LIN {X 0.048,Y -167.704,Z 705.356,A 0.000,B 0.000,C 90.000,E1 244.101} C_DIS
LIN {X 0.061,Y -166.391,Z 705.347,A 0.000,B 0.000,C 90.000,E1 242.359} C_DIS
LIN {X 0.052,Y -163.118,Z 705.327,A 0.000,B 0.000,C 90.000,E1 238.869} C_DIS
LIN {X 0.102,Y -161.067,Z 705.313,A 0.000,B 0.000,C 90.000,E1 236.215} C_DIS
LIN {X -0.010,Y -157.800,Z 705.293,A 0.000,B 0.000,C 90.000,E1 232.718} C_DIS
LIN {X -0.072,Y -155.836,Z 705.278,A 0.000,B 0.000,C 90.000,E1 230.070} C_DIS
LIN {X -0.015,Y -152.086,Z 705.253,A 0.000,B 0.000,C 90.000,E1 225.567} C_DIS
LIN {X 0.004,Y -150.337,Z 705.238,A 0.000,B 0.000,C 90.000,E1 222.852} C_DIS
LIN {X 0.025,Y -147.076,Z 705.213,A 0.000,B 0.000,C 90.000,E1 218.302} C_DIS
LIN {X -0.071,Y -145.650,Z 705.198,A 0.000,B 0.000,C 90.000,E1 215.598} C_DIS
LIN {X -0.067,Y -143.032,Z 705.172,A 0.000,B 0.000,C 90.000,E1 211.003} C_DIS
LIN {X 0.059,Y -141.657,Z 705.152,A 0.000,B 0.000,C 90.000,E1 207.257} C_DIS
LIN {X -0.022,Y -139.447,Z 705.115,A 0.000,B 0.000,C 90.000,E1 200.791} C_DIS
LIN {X 0.031,Y -139.180,Z 705.105,A 0.000,B 0.000,C 90.000,E1 198.906} C_DIS
LIN {X 0.059,Y -138.320,Z 705.053,A 0.000,B 0.000,C 90.000,E1 189.557} C_DIS
LIN {X 0.069,Y -139.465,Z 705.007,A 0.000,B 0.000,C 90.000,E1 181.146} C_DIS
LIN {X 0.010,Y -141.029,Z 704.975,A 0.000,B 0.000,C 90.000,E1 175.584} C_DIS
LIN {X -0.036,Y -142.396,Z 704.960,A 0.000,B 0.000,C 90.000,E1 172.818} C_DIS
LIN {X 0.026,Y -144.628,Z 704.934,A 0.000,B 0.000,C 90.000,E1 168.173} C_DIS
LIN {X -0.055,Y -147.823,Z 704.909,A 0.000,B 0.000,C 90.000,E1 163.614} C_DIS
LIN {X 0.031,Y -150.514,Z 704.889,A 0.000,B 0.000,C 90.000,E1 159.934} C_DIS
LIN {X 0.052,Y -153.976,Z 704.868,A 0.000,B 0.000,C 90.000,E1 156.305} C_DIS
LIN {X -0.027,Y -157.387,Z 704.849,A 0.000,B 0.000,C 90.000,E1 152.743} C_DIS
LIN {X -0.085,Y -161.592,Z 704.829,A 0.000,B 0.000,C 90.000,E1 149.203} C_DIS
LIN {X -0.075,Y -165.789,Z 704.809,A 0.000,B 0.000,C 90.000,E1 145.674} C_DIS
LIN {X -0.089,Y -170.750,Z 704.790,A 0.000,B 0.000,C 90.000,E1 142.190} C_DIS
LIN {X 0.069,Y -175.622,Z 704.771,A 0.000,B 0.000,C 90.000,E1 138.690} C_DIS
LIN {X -0.062,Y -181.238,Z 704.752,A 0.000,B 0.000,C 90.000,E1 135.324} C_DIS
LIN {X 0.069,Y -186.708,Z 704.733,A 0.000,B 0.000,C 90.000,E1 131.919} C_DIS
LIN {X 0.013,Y -191.370,Z 704.719,A 0.000,B 0.000,C 90.000,E1 129.402} C_DIS
LIN {X -0.035,Y -289.460,Z 704.719,A 0.000,B 0.000,C 90.000,E1 129.402} C_DIS
LIN {X 0.082,Y -291.032,Z 704.719,A 0.000,B 0.000,C 90.000,E1 129.358} C_DIS
LIN {X -0.059,Y -295.409,Z 704.718,A 0.000,B 0.000,C 90.000,E1 129.197} C_DIS
LIN {X 0.028,Y -297.779,Z 704.717,A 0.000,B 0.000,C 90.000,E1 128.991} C_DIS
LIN {X -0.027,Y -301.000,Z 704.715,A 0.000,B 0.000,C 90.000,E1 128.624} C_DIS
LIN {X -0.016,Y -302.956,Z 704.713,A 0.000,B 0.000,C 90.000,E1 128.302} C_DIS
LIN {X 0.045,Y -304.482,Z 704.711,A 0.000,B 0.000,C 90.000,E1 127.971} C_DIS
LIN {X 0.006,Y -305.724,Z 704.709,A 0.000,B 0.000,C 90.000,E1 127.649} C_DIS
LIN {X 0.198,Y -317.437,Z 704.687,A 0.000,B 0.000,C 90.000,E1 123.706} C_DIS
LIN {X -0.041,Y -327.590,Z 704.672,A 0.000,B 0.000,C 90.000,E1 120.875} C_DIS
LIN {X 0.128,Y -339.075,Z 704.656,A 0.000,B 0.000,C 90.000,E1 118.025} C_DIS
LIN {X -0.014,Y -352.001,Z 704.640,A 0.000,B 0.000,C 90.000,E1 115.283} C_DIS
LIN {X -0.151,Y -364.788,Z 704.627,A 0.000,B 0.000,C 90.000,E1 112.898} C_DIS
LIN {X 0.230,Y -378.895,Z 704.614,A 0.000,B 0.000,C 90.000,E1 110.482} C_DIS
LIN {X -0.150,Y -394.422,Z 704.601,A 0.000,B 0.000,C 90.000,E1 108.236} C_DIS
LIN {X -0.016,Y -411.481,Z 704.589,A 0.000,B 0.000,C 90.000,E1 105.969} C_DIS
LIN {X 0.046,Y -430.198,Z 704.577,A 0.000,B 0.000,C 90.000,E1 103.772} C_DIS
LIN {X -0.104,Y -450.192,Z 704.565,A 0.000,B 0.000,C 90.000,E1 101.715} C_DIS
LIN {X 0.076,Y -468.132,Z 704.556,A 0.000,B 0.000,C 90.000,E1 100.018} C_DIS
LIN {X 0.038,Y -470.302,Z 704.554,A 0.000,B 0.000,C 90.000,E1 99.792} C_DIS
LIN {X -0.111,Y -472.091,Z 704.553,A 0.000,B 0.000,C 90.000,E1 99.557} C_DIS
LIN {X 0.203,Y -473.434,Z 704.552,A 0.000,B 0.000,C 90.000,E1 99.265} C_DIS
LIN {X -0.154,Y -475.119,Z 704.549,A 0.000,B 0.000,C 90.000,E1 98.803} C_DIS
LIN {X 0.036,Y -475.734,Z 704.546,A 0.000,B 0.000,C 90.000,E1 98.276} C_DIS
LIN {X 0.167,Y -475.383,Z 704.543,A 0.000,B 0.000,C 90.000,E1 97.757} C_DIS
LIN {X -0.170,Y -474.017,Z 704.540,A 0.000,B 0.000,C 90.000,E1 97.296} C_DIS
LIN {X 0.104,Y -472.884,Z 704.539,A 0.000,B 0.000,C 90.000,E1 97.011} C_DIS
LIN {X -0.182,Y -469.662,Z 704.536,A 0.000,B 0.000,C 90.000,E1 96.543} C_DIS
LIN {X -0.116,Y -451.783,Z 704.521,A 0.000,B 0.000,C 90.000,E1 93.726} C_DIS
LIN {X 0.073,Y -437.091,Z 704.506,A 0.000,B 0.000,C 90.000,E1 91.088} C_DIS
LIN {X 0.141,Y -428.050,Z 704.497,A 0.000,B 0.000,C 90.000,E1 89.484} C_DIS
LIN {X 0.059,Y -418.745,Z 704.488,A 0.000,B 0.000,C 90.000,E1 87.879} C_DIS
LIN {X -0.107,Y -407.783,Z 704.478,A 0.000,B 0.000,C 90.000,E1 85.988} C_DIS
LIN {X -0.039,Y -396.834,Z 704.467,A 0.000,B 0.000,C 90.000,E1 84.033} C_DIS
LIN {X -0.045,Y -381.422,Z 704.451,A 0.000,B 0.000,C 90.000,E1 81.197} C_DIS
LIN {X 0.006,Y -368.132,Z 704.437,A 0.000,B 0.000,C 90.000,E1 78.578} C_DIS
LIN {X -0.201,Y -353.954,Z 704.420,A 0.000,B 0.000,C 90.000,E1 75.644} C_DIS
LIN {X -0.131,Y -340.345,Z 704.403,A 0.000,B 0.000,C 90.000,E1 72.598} C_DIS
LIN {X -0.098,Y -329.846,Z 704.389,A 0.000,B 0.000,C 90.000,E1 70.115} C_DIS
LIN {X 0.087,Y -317.557,Z 704.372,A 0.000,B 0.000,C 90.000,E1 66.922} C_DIS
LIN {X 0.085,Y -307.850,Z 704.356,A 0.000,B 0.000,C 90.000,E1 64.024} C_DIS
LIN {X -0.151,Y -298.135,Z 704.338,A 0.000,B 0.000,C 90.000,E1 60.795} C_DIS
LIN {X -0.097,Y -289.035,Z 704.319,A 0.000,B 0.000,C 90.000,E1 57.454} C_DIS
LIN {X -0.026,Y -282.114,Z 704.304,A 0.000,B 0.000,C 90.000,E1 54.736} C_DIS
LIN {X -0.020,Y -277.046,Z 704.293,A 0.000,B 0.000,C 90.000,E1 52.683} C_DIS
LIN {X 0.048,Y -271.812,Z 704.281,A 0.000,B 0.000,C 90.000,E1 50.598} C_DIS
LIN {X -0.057,Y -266.456,Z 704.270,A 0.000,B 0.000,C 90.000,E1 48.528} C_DIS
LIN {X 0.116,Y -260.753,Z 704.258,A 0.000,B 0.000,C 90.000,E1 46.377} C_DIS
LIN {X -0.019,Y -254.912,Z 704.246,A 0.000,B 0.000,C 90.000,E1 44.271} C_DIS
LIN {X 0.105,Y -248.878,Z 704.234,A 0.000,B 0.000,C 90.000,E1 42.081} C_DIS
LIN {X -0.052,Y -242.729,Z 704.222,A 0.000,B 0.000,C 90.000,E1 39.930} C_DIS
LIN {X -0.017,Y -232.750,Z 704.201,A 0.000,B 0.000,C 90.000,E1 36.217} C_DIS
LIN {X 0.054,Y -223.570,Z 704.180,A 0.000,B 0.000,C 90.000,E1 32.418} C_DIS
LIN {X 0.088,Y -216.951,Z 704.163,A 0.000,B 0.000,C 90.000,E1 29.333} C_DIS
LIN {X 0.021,Y -211.168,Z 704.146,A 0.000,B 0.000,C 90.000,E1 26.232} C_DIS
LIN {X 0.009,Y -206.116,Z 704.128,A 0.000,B 0.000,C 90.000,E1 23.078} C_DIS
LIN {X 0.001,Y -200.975,Z 704.106,A 0.000,B 0.000,C 90.000,E1 19.087} C_DIS
LIN {X -0.045,Y -197.005,Z 704.084,A 0.000,B 0.000,C 90.000,E1 15.064} C_DIS
LIN {X 0.079,Y -193.660,Z 704.056,A 0.000,B 0.000,C 90.000,E1 10.141} C_DIS
LIN {X 0.021,Y -191.501,Z 704.011,A 0.000,B 0.000,C 90.000,E1 1.949} C_DIS
LIN {X -0.072,Y -193.432,Z 703.965,A 0.000,B 0.000,C 90.000,E1 353.799} C_DIS
LIN {X -0.003,Y -196.450,Z 703.938,A 0.000,B 0.000,C 90.000,E1 348.870} C_DIS
LIN {X -0.015,Y -200.116,Z 703.916,A 0.000,B 0.000,C 90.000,E1 344.810} C_DIS
LIN {X -0.030,Y -204.725,Z 703.893,A 0.000,B 0.000,C 90.000,E1 340.786} C_DIS
LIN {X -0.012,Y -210.168,Z 703.871,A 0.000,B 0.000,C 90.000,E1 336.794} C_DIS
LIN {X -0.073,Y -216.346,Z 703.849,A 0.000,B 0.000,C 90.000,E1 332.871} C_DIS
LIN {X 0.070,Y -223.240,Z 703.828,A 0.000,B 0.000,C 90.000,E1 328.948} C_DIS
LIN {X 0.008,Y -230.745,Z 703.806,A 0.000,B 0.000,C 90.000,E1 325.135} C_DIS
LIN {X -0.035,Y -238.853,Z 703.785,A 0.000,B 0.000,C 90.000,E1 321.376} C_DIS
LIN {X 0.120,Y -247.875,Z 703.765,A 0.000,B 0.000,C 90.000,E1 317.634} C_DIS
LIN {X -0.006,Y -257.951,Z 703.745,A 0.000,B 0.000,C 90.000,E1 314.028} C_DIS
LIN {X 0.048,Y -269.153,Z 703.725,A 0.000,B 0.000,C 90.000,E1 310.458} C_DIS
LIN {X 0.082,Y -280.335,Z 703.707,A 0.000,B 0.000,C 90.000,E1 307.317} C_DIS
LIN {X 0.085,Y -294.112,Z 703.688,A 0.000,B 0.000,C 90.000,E1 303.913} C_DIS
LIN {X 0.115,Y -309.286,Z 703.670,A 0.000,B 0.000,C 90.000,E1 300.590} C_DIS
LIN {X -0.011,Y -322.591,Z 703.656,A 0.000,B 0.000,C 90.000,E1 298.025} C_DIS
LIN {X -0.155,Y -340.634,Z 703.638,A 0.000,B 0.000,C 90.000,E1 294.899} C_DIS
LIN {X 0.090,Y -356.064,Z 703.625,A 0.000,B 0.000,C 90.000,E1 292.408} C_DIS
LIN {X -0.208,Y -372.171,Z 703.611,A 0.000,B 0.000,C 90.000,E1 290.066} C_DIS
LIN {X 0.112,Y -390.115,Z 703.598,A 0.000,B 0.000,C 90.000,E1 287.692} C_DIS
LIN {X -0.117,Y -404.103,Z 703.589,A 0.000,B 0.000,C 90.000,E1 286.024} C_DIS
LIN {X -0.100,Y -417.902,Z 703.580,A 0.000,B 0.000,C 90.000,E1 284.356} C_DIS
LIN {X -0.206,Y -429.223,Z 703.572,A 0.000,B 0.000,C 90.000,E1 283.008} C_DIS
LIN {X 0.093,Y -437.971,Z 703.566,A 0.000,B 0.000,C 90.000,E1 281.895} C_DIS
LIN {X -0.136,Y -448.227,Z 703.559,A 0.000,B 0.000,C 90.000,E1 280.602} C_DIS
LIN {X -0.022,Y -464.309,Z 703.547,A 0.000,B 0.000,C 90.000,E1 278.511} C_DIS
LIN {X 0.115,Y -472.091,Z 703.542,A 0.000,B 0.000,C 90.000,E1 277.473} C_DIS
LIN {X 0.074,Y -477.214,Z 703.537,A 0.000,B 0.000,C 90.000,E1 276.720} C_DIS
LIN {X 0.213,Y -480.183,Z 703.535,A 0.000,B 0.000,C 90.000,E1 276.201} C_DIS
LIN {X -0.110,Y -482.767,Z 703.532,A 0.000,B 0.000,C 90.000,E1 275.739} C_DIS
LIN {X 0.061,Y -484.885,Z 703.529,A 0.000,B 0.000,C 90.000,E1 275.220} C_DIS
LIN {X 0.246,Y -486.541,Z 703.526,A 0.000,B 0.000,C 90.000,E1 274.702} C_DIS
LIN {X -0.087,Y -487.760,Z 703.523,A 0.000,B 0.000,C 90.000,E1 274.245} C_DIS
LIN {X 0.113,Y -488.620,Z 703.521,A 0.000,B 0.000,C 90.000,E1 273.726} C_DIS
LIN {X -0.200,Y -489.020,Z 703.518,A 0.000,B 0.000,C 90.000,E1 273.269} C_DIS
LIN {X 0.008,Y -489.135,Z 703.515,A 0.000,B 0.000,C 90.000,E1 272.751} C_DIS
LIN {X 0.194,Y -488.868,Z 703.513,A 0.000,B 0.000,C 90.000,E1 272.236} C_DIS
LIN {X -0.089,Y -488.311,Z 703.510,A 0.000,B 0.000,C 90.000,E1 271.776} C_DIS
LIN {X 0.096,Y -487.341,Z 703.507,A 0.000,B 0.000,C 90.000,E1 271.260} C_DIS
LIN {X -0.207,Y -485.976,Z 703.504,A 0.000,B 0.000,C 90.000,E1 270.802} C_DIS
LIN {X -0.028,Y -484.154,Z 703.502,A 0.000,B 0.000,C 90.000,E1 270.286} C_DIS
LIN {X 0.143,Y -481.763,Z 703.499,A 0.000,B 0.000,C 90.000,E1 269.771} C_DIS
LIN {X -0.184,Y -478.781,Z 703.496,A 0.000,B 0.000,C 90.000,E1 269.312} C_DIS
LIN {X -0.048,Y -474.923,Z 703.493,A 0.000,B 0.000,C 90.000,E1 268.797} C_DIS
LIN {X 0.066,Y -470.084,Z 703.490,A 0.000,B 0.000,C 90.000,E1 268.282} C_DIS
LIN {X -0.053,Y -467.317,Z 703.489,A 0.000,B 0.000,C 90.000,E1 268.051} C_DIS
LIN {X -0.029,Y -461.152,Z 703.487,A 0.000,B 0.000,C 90.000,E1 267.593} C_DIS
LIN {X 0.122,Y -457.794,Z 703.485,A 0.000,B 0.000,C 90.000,E1 267.364} C_DIS
LIN {X 0.064,Y -454.502,Z 703.484,A 0.000,B 0.000,C 90.000,E1 267.192} C_DIS
LIN {X -0.179,Y -447.359,Z 703.483,A 0.000,B 0.000,C 90.000,E1 266.906} C_DIS
LIN {X 0.142,Y -440.044,Z 703.481,A 0.000,B 0.000,C 90.000,E1 266.617} C_DIS
LIN {X -0.018,Y -431.920,Z 703.480,A 0.000,B 0.000,C 90.000,E1 266.445} C_DIS
LIN {X -0.208,Y -426.165,Z 703.480,A 0.000,B 0.000,C 90.000,E1 266.388} C_DIS
LIN {X 0.159,Y -417.344,Z 703.479,A 0.000,B 0.000,C 90.000,E1 266.274} C_DIS
LIN {X 0.048,Y -180.934,Z 703.479,A 0.000,B 0.000,C 90.000,E1 266.274} C_DIS
LIN {X 0.080,Y -180.714,Z 703.470,A 0.000,B 0.000,C 90.000,E1 264.552} C_DIS
LIN {X -0.002,Y -178.800,Z 703.442,A 0.000,B 0.000,C 90.000,E1 259.511} C_DIS
LIN {X 0.075,Y -175.846,Z 703.413,A 0.000,B 0.000,C 90.000,E1 254.393} C_DIS
LIN {X 0.075,Y -172.037,Z 703.385,A 0.000,B 0.000,C 90.000,E1 249.263} C_DIS
LIN {X 0.051,Y -171.469,Z 703.380,A 0.000,B 0.000,C 90.000,E1 248.411} C_DIS
LIN {X 0.030,Y -167.700,Z 703.356,A 0.000,B 0.000,C 90.000,E1 244.101} C_DIS
LIN {X 0.043,Y -166.385,Z 703.346,A 0.000,B 0.000,C 90.000,E1 242.359} C_DIS
LIN {X 0.035,Y -163.113,Z 703.327,A 0.000,B 0.000,C 90.000,E1 238.869} C_DIS
LIN {X 0.085,Y -161.062,Z 703.313,A 0.000,B 0.000,C 90.000,E1 236.215} C_DIS
LIN {X -0.027,Y -157.795,Z 703.293,A 0.000,B 0.000,C 90.000,E1 232.718} C_DIS
LIN {X 0.012,Y -155.832,Z 703.278,A 0.000,B 0.000,C 90.000,E1 230.033} C_DIS
LIN {X -0.031,Y -152.082,Z 703.253,A 0.000,B 0.000,C 90.000,E1 225.567} C_DIS
LIN {X -0.013,Y -150.333,Z 703.238,A 0.000,B 0.000,C 90.000,E1 222.852} C_DIS
LIN {X 0.008,Y -147.073,Z 703.213,A 0.000,B 0.000,C 90.000,E1 218.302} C_DIS
LIN {X -0.088,Y -145.647,Z 703.198,A 0.000,B 0.000,C 90.000,E1 215.598} C_DIS
LIN {X -0.083,Y -143.029,Z 703.172,A 0.000,B 0.000,C 90.000,E1 211.003} C_DIS
LIN {X 0.044,Y -141.655,Z 703.152,A 0.000,B 0.000,C 90.000,E1 207.257} C_DIS
LIN {X -0.037,Y -139.445,Z 703.115,A 0.000,B 0.000,C 90.000,E1 200.791} C_DIS
LIN {X 0.016,Y -139.179,Z 703.105,A 0.000,B 0.000,C 90.000,E1 198.906} C_DIS
LIN {X 0.044,Y -138.320,Z 703.053,A 0.000,B 0.000,C 90.000,E1 189.557} C_DIS
LIN {X 0.053,Y -139.467,Z 703.006,A 0.000,B 0.000,C 90.000,E1 181.146} C_DIS
LIN {X -0.006,Y -141.032,Z 702.975,A 0.000,B 0.000,C 90.000,E1 175.584} C_DIS
LIN {X -0.052,Y -142.399,Z 702.960,A 0.000,B 0.000,C 90.000,E1 172.818} C_DIS
LIN {X 0.011,Y -144.631,Z 702.934,A 0.000,B 0.000,C 90.000,E1 168.173} C_DIS
LIN {X 0.071,Y -147.827,Z 702.909,A 0.000,B 0.000,C 90.000,E1 163.559} C_DIS
LIN {X 0.016,Y -150.520,Z 702.889,A 0.000,B 0.000,C 90.000,E1 159.934} C_DIS
LIN {X 0.035,Y -153.982,Z 702.868,A 0.000,B 0.000,C 90.000,E1 156.305} C_DIS
LIN {X -0.045,Y -157.394,Z 702.849,A 0.000,B 0.000,C 90.000,E1 152.743} C_DIS
LIN {X 0.036,Y -161.600,Z 702.829,A 0.000,B 0.000,C 90.000,E1 149.154} C_DIS
LIN {X -0.092,Y -165.796,Z 702.809,A 0.000,B 0.000,C 90.000,E1 145.674} C_DIS
LIN {X 0.028,Y -170.759,Z 702.790,A 0.000,B 0.000,C 90.000,E1 142.145} C_DIS
LIN {X 0.051,Y -175.632,Z 702.771,A 0.000,B 0.000,C 90.000,E1 138.690} C_DIS
LIN {X -0.080,Y -181.247,Z 702.752,A 0.000,B 0.000,C 90.000,E1 135.324} C_DIS
LIN {X 0.050,Y -186.718,Z 702.733,A 0.000,B 0.000,C 90.000,E1 131.919} C_DIS
LIN {X 0.053,Y -191.351,Z 702.719,A 0.000,B 0.000,C 90.000,E1 129.402} C_DIS
LIN {X 0.044,Y -289.167,Z 702.719,A 0.000,B 0.000,C 90.000,E1 129.402} C_DIS
LIN {X 0.053,Y -291.778,Z 702.719,A 0.000,B 0.000,C 90.000,E1 129.358} C_DIS
LIN {X -0.089,Y -295.650,Z 702.718,A 0.000,B 0.000,C 90.000,E1 129.197} C_DIS
LIN {X -0.002,Y -297.932,Z 702.717,A 0.000,B 0.000,C 90.000,E1 128.991} C_DIS
LIN {X -0.058,Y -301.080,Z 702.715,A 0.000,B 0.000,C 90.000,E1 128.624} C_DIS
LIN {X -0.074,Y -303.031,Z 702.713,A 0.000,B 0.000,C 90.000,E1 128.302} C_DIS
LIN {X -0.040,Y -304.551,Z 702.711,A 0.000,B 0.000,C 90.000,E1 127.971} C_DIS
LIN {X -0.081,Y -305.766,Z 702.709,A 0.000,B 0.000,C 90.000,E1 127.649} C_DIS
LIN {X 0.109,Y -317.469,Z 702.687,A 0.000,B 0.000,C 90.000,E1 123.706} C_DIS
LIN {X -0.131,Y -327.628,Z 702.671,A 0.000,B 0.000,C 90.000,E1 120.875} C_DIS
LIN {X 0.035,Y -339.121,Z 702.656,A 0.000,B 0.000,C 90.000,E1 118.025} C_DIS
LIN {X -0.107,Y -352.054,Z 702.640,A 0.000,B 0.000,C 90.000,E1 115.283} C_DIS
LIN {X 0.088,Y -364.850,Z 702.627,A 0.000,B 0.000,C 90.000,E1 112.845} C_DIS
LIN {X 0.132,Y -378.965,Z 702.614,A 0.000,B 0.000,C 90.000,E1 110.482} C_DIS
LIN {X 0.124,Y -394.501,Z 702.601,A 0.000,B 0.000,C 90.000,E1 108.181} C_DIS
LIN {X -0.119,Y -411.570,Z 702.589,A 0.000,B 0.000,C 90.000,E1 105.969} C_DIS
LIN {X -0.060,Y -430.298,Z 702.576,A 0.000,B 0.000,C 90.000,E1 103.772} C_DIS
LIN {X -0.206,Y -450.295,Z 702.565,A 0.000,B 0.000,C 90.000,E1 101.715} C_DIS
LIN {X -0.023,Y -468.237,Z 702.556,A 0.000,B 0.000,C 90.000,E1 100.018} C_DIS
LIN {X -0.061,Y -470.396,Z 702.554,A 0.000,B 0.000,C 90.000,E1 99.792} C_DIS
LIN {X -0.211,Y -472.176,Z 702.553,A 0.000,B 0.000,C 90.000,E1 99.557} C_DIS
LIN {X 0.104,Y -473.513,Z 702.552,A 0.000,B 0.000,C 90.000,E1 99.265} C_DIS
LIN {X -0.253,Y -475.188,Z 702.549,A 0.000,B 0.000,C 90.000,E1 98.803} C_DIS
LIN {X -0.062,Y -475.795,Z 702.546,A 0.000,B 0.000,C 90.000,E1 98.276} C_DIS
LIN {X 0.069,Y -475.436,Z 702.543,A 0.000,B 0.000,C 90.000,E1 97.757} C_DIS
LIN {X 0.203,Y -474.060,Z 702.540,A 0.000,B 0.000,C 90.000,E1 97.239} C_DIS
LIN {X 0.064,Y -472.922,Z 702.539,A 0.000,B 0.000,C 90.000,E1 97.004} C_DIS
LIN {X 0.188,Y -469.694,Z 702.536,A 0.000,B 0.000,C 90.000,E1 96.486} C_DIS
LIN {X -0.208,Y -451.768,Z 702.521,A 0.000,B 0.000,C 90.000,E1 93.726} C_DIS
LIN {X -0.016,Y -437.088,Z 702.506,A 0.000,B 0.000,C 90.000,E1 91.088} C_DIS
LIN {X 0.054,Y -428.082,Z 702.497,A 0.000,B 0.000,C 90.000,E1 89.484} C_DIS
LIN {X 0.081,Y -417.200,Z 702.487,A 0.000,B 0.000,C 90.000,E1 87.593} C_DIS
LIN {X -0.089,Y -406.241,Z 702.476,A 0.000,B 0.000,C 90.000,E1 85.698} C_DIS
LIN {X -0.118,Y -396.864,Z 702.467,A 0.000,B 0.000,C 90.000,E1 84.033} C_DIS
LIN {X -0.120,Y -381.467,Z 702.451,A 0.000,B 0.000,C 90.000,E1 81.197} C_DIS
LIN {X -0.065,Y -368.205,Z 702.436,A 0.000,B 0.000,C 90.000,E1 78.578} C_DIS
LIN {X 0.075,Y -354.027,Z 702.420,A 0.000,B 0.000,C 90.000,E1 75.589} C_DIS
LIN {X 0.131,Y -340.470,Z 702.403,A 0.000,B 0.000,C 90.000,E1 72.543} C_DIS
LIN {X 0.155,Y -329.993,Z 702.389,A 0.000,B 0.000,C 90.000,E1 70.061} C_DIS
LIN {X 0.038,Y -317.748,Z 702.372,A 0.000,B 0.000,C 90.000,E1 66.922} C_DIS
LIN {X 0.042,Y -308.053,Z 702.356,A 0.000,B 0.000,C 90.000,E1 64.024} C_DIS
LIN {X -0.187,Y -298.358,Z 702.338,A 0.000,B 0.000,C 90.000,E1 60.795} C_DIS
LIN {X -0.124,Y -289.286,Z 702.319,A 0.000,B 0.000,C 90.000,E1 57.454} C_DIS
LIN {X -0.046,Y -282.387,Z 702.304,A 0.000,B 0.000,C 90.000,E1 54.736} C_DIS
LIN {X -0.036,Y -277.320,Z 702.293,A 0.000,B 0.000,C 90.000,E1 52.683} C_DIS
LIN {X 0.038,Y -272.122,Z 702.281,A 0.000,B 0.000,C 90.000,E1 50.598} C_DIS
LIN {X -0.060,Y -266.768,Z 702.270,A 0.000,B 0.000,C 90.000,E1 48.528} C_DIS
LIN {X 0.118,Y -261.057,Z 702.258,A 0.000,B 0.000,C 90.000,E1 46.377} C_DIS
LIN {X -0.012,Y -255.182,Z 702.246,A 0.000,B 0.000,C 90.000,E1 44.271} C_DIS
LIN {X -0.067,Y -249.164,Z 702.234,A 0.000,B 0.000,C 90.000,E1 42.123} C_DIS
LIN {X -0.034,Y -242.980,Z 702.222,A 0.000,B 0.000,C 90.000,E1 39.930} C_DIS
LIN {X 0.006,Y -232.950,Z 702.201,A 0.000,B 0.000,C 90.000,E1 36.217} C_DIS
LIN {X 0.082,Y -223.756,Z 702.180,A 0.000,B 0.000,C 90.000,E1 32.418} C_DIS
LIN {X 0.121,Y -217.115,Z 702.163,A 0.000,B 0.000,C 90.000,E1 29.333} C_DIS
LIN {X 0.057,Y -211.333,Z 702.146,A 0.000,B 0.000,C 90.000,E1 26.232} C_DIS
LIN {X 0.048,Y -206.277,Z 702.128,A 0.000,B 0.000,C 90.000,E1 23.078} C_DIS
LIN {X 0.044,Y -201.134,Z 702.106,A 0.000,B 0.000,C 90.000,E1 19.087} C_DIS
LIN {X 0.003,Y -197.160,Z 702.084,A 0.000,B 0.000,C 90.000,E1 15.064} C_DIS
LIN {X -0.059,Y -193.825,Z 702.057,A 0.000,B 0.000,C 90.000,E1 10.197} C_DIS
LIN {X 0.082,Y -191.648,Z 702.011,A 0.000,B 0.000,C 90.000,E1 1.949} C_DIS
LIN {X -0.066,Y -193.542,Z 701.965,A 0.000,B 0.000,C 90.000,E1 353.799} C_DIS
LIN {X 0.008,Y -196.562,Z 701.938,A 0.000,B 0.000,C 90.000,E1 348.870} C_DIS
LIN {X -0.001,Y -200.208,Z 701.916,A 0.000,B 0.000,C 90.000,E1 344.810} C_DIS
LIN {X -0.013,Y -204.805,Z 701.893,A 0.000,B 0.000,C 90.000,E1 340.786} C_DIS
LIN {X 0.008,Y -210.234,Z 701.871,A 0.000,B 0.000,C 90.000,E1 336.794} C_DIS
LIN {X -0.050,Y -216.404,Z 701.849,A 0.000,B 0.000,C 90.000,E1 332.871} C_DIS
LIN {X -0.097,Y -223.286,Z 701.828,A 0.000,B 0.000,C 90.000,E1 328.997} C_DIS
LIN {X 0.035,Y -230.773,Z 701.806,A 0.000,B 0.000,C 90.000,E1 325.135} C_DIS
LIN {X -0.006,Y -238.876,Z 701.785,A 0.000,B 0.000,C 90.000,E1 321.376} C_DIS
LIN {X -0.032,Y -247.896,Z 701.765,A 0.000,B 0.000,C 90.000,E1 317.676} C_DIS
LIN {X 0.028,Y -257.967,Z 701.745,A 0.000,B 0.000,C 90.000,E1 314.028} C_DIS
LIN {X 0.084,Y -269.167,Z 701.725,A 0.000,B 0.000,C 90.000,E1 310.458} C_DIS
LIN {X -0.103,Y -280.348,Z 701.707,A 0.000,B 0.000,C 90.000,E1 307.363} C_DIS
LIN {X 0.124,Y -294.121,Z 701.689,A 0.000,B 0.000,C 90.000,E1 303.913} C_DIS
LIN {X 0.157,Y -309.292,Z 701.670,A 0.000,B 0.000,C 90.000,E1 300.590} C_DIS
LIN {X 0.033,Y -322.585,Z 701.656,A 0.000,B 0.000,C 90.000,E1 298.025} C_DIS
LIN {X -0.110,Y -340.598,Z 701.638,A 0.000,B 0.000,C 90.000,E1 294.899} C_DIS
LIN {X -0.155,Y -357.955,Z 701.623,A 0.000,B 0.000,C 90.000,E1 292.153} C_DIS
LIN {X -0.160,Y -372.051,Z 701.611,A 0.000,B 0.000,C 90.000,E1 290.066} C_DIS
LIN {X 0.014,Y -387.646,Z 701.600,A 0.000,B 0.000,C 90.000,E1 288.000} C_DIS
LIN {X -0.146,Y -401.637,Z 701.591,A 0.000,B 0.000,C 90.000,E1 286.315} C_DIS
LIN {X 0.223,Y -415.433,Z 701.581,A 0.000,B 0.000,C 90.000,E1 284.592} C_DIS
LIN {X 0.093,Y -426.792,Z 701.574,A 0.000,B 0.000,C 90.000,E1 283.244} C_DIS
LIN {X -0.057,Y -435.628,Z 701.568,A 0.000,B 0.000,C 90.000,E1 282.187} C_DIS
LIN {X 0.109,Y -446.003,Z 701.560,A 0.000,B 0.000,C 90.000,E1 280.838} C_DIS
LIN {X 0.184,Y -462.066,Z 701.549,A 0.000,B 0.000,C 90.000,E1 278.746} C_DIS
LIN {X -0.102,Y -470.009,Z 701.543,A 0.000,B 0.000,C 90.000,E1 277.757} C_DIS
LIN {X -0.162,Y -475.402,Z 701.539,A 0.000,B 0.000,C 90.000,E1 277.004} C_DIS
LIN {X -0.039,Y -478.609,Z 701.536,A 0.000,B 0.000,C 90.000,E1 276.486} C_DIS
LIN {X -0.083,Y -482.625,Z 701.532,A 0.000,B 0.000,C 90.000,E1 275.739} C_DIS
LIN {X 0.087,Y -484.742,Z 701.529,A 0.000,B 0.000,C 90.000,E1 275.220} C_DIS
LIN {X -0.213,Y -486.412,Z 701.526,A 0.000,B 0.000,C 90.000,E1 274.759} C_DIS
LIN {X -0.063,Y -487.677,Z 701.524,A 0.000,B 0.000,C 90.000,E1 274.245} C_DIS
LIN {X 0.136,Y -488.485,Z 701.521,A 0.000,B 0.000,C 90.000,E1 273.726} C_DIS
LIN {X -0.177,Y -488.916,Z 701.518,A 0.000,B 0.000,C 90.000,E1 273.269} C_DIS
LIN {X 0.030,Y -489.010,Z 701.515,A 0.000,B 0.000,C 90.000,E1 272.751} C_DIS
LIN {X 0.216,Y -488.794,Z 701.513,A 0.000,B 0.000,C 90.000,E1 272.236} C_DIS
LIN {X -0.069,Y -488.232,Z 701.510,A 0.000,B 0.000,C 90.000,E1 271.776} C_DIS
LIN {X 0.117,Y -487.276,Z 701.507,A 0.000,B 0.000,C 90.000,E1 271.260} C_DIS
LIN {X -0.186,Y -485.918,Z 701.504,A 0.000,B 0.000,C 90.000,E1 270.802} C_DIS
LIN {X -0.007,Y -484.089,Z 701.502,A 0.000,B 0.000,C 90.000,E1 270.286} C_DIS
LIN {X 0.162,Y -481.745,Z 701.499,A 0.000,B 0.000,C 90.000,E1 269.771} C_DIS
LIN {X -0.166,Y -478.739,Z 701.496,A 0.000,B 0.000,C 90.000,E1 269.312} C_DIS
LIN {X -0.029,Y -474.902,Z 701.493,A 0.000,B 0.000,C 90.000,E1 268.797} C_DIS
LIN {X 0.084,Y -470.050,Z 701.491,A 0.000,B 0.000,C 90.000,E1 268.282} C_DIS
LIN {X -0.023,Y -467.314,Z 701.489,A 0.000,B 0.000,C 90.000,E1 268.051} C_DIS
LIN {X 0.007,Y -461.260,Z 701.487,A 0.000,B 0.000,C 90.000,E1 267.593} C_DIS
LIN {X 0.156,Y -457.864,Z 701.485,A 0.000,B 0.000,C 90.000,E1 267.364} C_DIS
LIN {X 0.059,Y -450.853,Z 701.483,A 0.000,B 0.000,C 90.000,E1 267.020} C_DIS
LIN {X 0.081,Y -443.504,Z 701.482,A 0.000,B 0.000,C 90.000,E1 266.731} C_DIS
LIN {X 0.125,Y -435.832,Z 701.481,A 0.000,B 0.000,C 90.000,E1 266.502} C_DIS
LIN {X -0.071,Y -431.766,Z 701.480,A 0.000,B 0.000,C 90.000,E1 266.445} C_DIS
LIN {X 0.165,Y -425.980,Z 701.480,A 0.000,B 0.000,C 90.000,E1 266.331} C_DIS
LIN {X 0.107,Y -417.182,Z 701.479,A 0.000,B 0.000,C 90.000,E1 266.274} C_DIS
LIN {X 0.026,Y -180.934,Z 701.479,A 0.000,B 0.000,C 90.000,E1 266.274} C_DIS
LIN {X 0.002,Y -180.906,Z 701.474,A 0.000,B 0.000,C 90.000,E1 265.412} C_DIS
LIN {X 0.059,Y -180.710,Z 701.470,A 0.000,B 0.000,C 90.000,E1 264.552} C_DIS
LIN {X -0.023,Y -178.797,Z 701.442,A 0.000,B 0.000,C 90.000,E1 259.511} C_DIS
LIN {X 0.054,Y -175.843,Z 701.413,A 0.000,B 0.000,C 90.000,E1 254.393} C_DIS
LIN {X 0.053,Y -172.033,Z 701.385,A 0.000,B 0.000,C 90.000,E1 249.263} C_DIS
LIN {X 0.030,Y -171.462,Z 701.380,A 0.000,B 0.000,C 90.000,E1 248.411} C_DIS
LIN {X 0.010,Y -167.694,Z 701.356,A 0.000,B 0.000,C 90.000,E1 244.101} C_DIS
LIN {X 0.024,Y -166.378,Z 701.346,A 0.000,B 0.000,C 90.000,E1 242.359} C_DIS
LIN {X 0.016,Y -163.107,Z 701.327,A 0.000,B 0.000,C 90.000,E1 238.869} C_DIS
LIN {X 0.066,Y -161.054,Z 701.312,A 0.000,B 0.000,C 90.000,E1 236.215} C_DIS
LIN {X 0.048,Y -157.789,Z 701.293,A 0.000,B 0.000,C 90.000,E1 232.683} C_DIS
LIN {X -0.008,Y -155.826,Z 701.278,A 0.000,B 0.000,C 90.000,E1 230.033} C_DIS
LIN {X -0.051,Y -152.077,Z 701.253,A 0.000,B 0.000,C 90.000,E1 225.567} C_DIS
LIN {X -0.032,Y -150.327,Z 701.238,A 0.000,B 0.000,C 90.000,E1 222.852} C_DIS
LIN {X -0.011,Y -147.068,Z 701.213,A 0.000,B 0.000,C 90.000,E1 218.302} C_DIS
LIN {X 0.097,Y -145.643,Z 701.198,A 0.000,B 0.000,C 90.000,E1 215.518} C_DIS
LIN {X 0.094,Y -143.026,Z 701.172,A 0.000,B 0.000,C 90.000,E1 210.924} C_DIS
LIN {X 0.025,Y -141.651,Z 701.151,A 0.000,B 0.000,C 90.000,E1 207.257} C_DIS
LIN {X -0.055,Y -139.444,Z 701.115,A 0.000,B 0.000,C 90.000,E1 200.791} C_DIS
LIN {X -0.003,Y -139.177,Z 701.105,A 0.000,B 0.000,C 90.000,E1 198.906} C_DIS
LIN {X 0.026,Y -138.319,Z 701.053,A 0.000,B 0.000,C 90.000,E1 189.557} C_DIS
LIN {X 0.035,Y -139.468,Z 701.006,A 0.000,B 0.000,C 90.000,E1 181.146} C_DIS
LIN {X -0.025,Y -141.035,Z 700.975,A 0.000,B 0.000,C 90.000,E1 175.584} C_DIS
LIN {X 0.071,Y -142.403,Z 700.960,A 0.000,B 0.000,C 90.000,E1 172.761} C_DIS
LIN {X -0.009,Y -144.636,Z 700.934,A 0.000,B 0.000,C 90.000,E1 168.173} C_DIS
LIN {X 0.052,Y -147.831,Z 700.909,A 0.000,B 0.000,C 90.000,E1 163.559} C_DIS
LIN {X -0.004,Y -150.526,Z 700.888,A 0.000,B 0.000,C 90.000,E1 159.934} C_DIS
LIN {X 0.015,Y -153.988,Z 700.868,A 0.000,B 0.000,C 90.000,E1 156.305} C_DIS
LIN {X -0.064,Y -157.402,Z 700.848,A 0.000,B 0.000,C 90.000,E1 152.743} C_DIS
LIN {X 0.016,Y -161.608,Z 700.829,A 0.000,B 0.000,C 90.000,E1 149.154} C_DIS
LIN {X -0.019,Y -165.805,Z 700.809,A 0.000,B 0.000,C 90.000,E1 145.642} C_DIS
LIN {X 0.007,Y -170.770,Z 700.790,A 0.000,B 0.000,C 90.000,E1 142.145} C_DIS
LIN {X 0.029,Y -175.642,Z 700.771,A 0.000,B 0.000,C 90.000,E1 138.690} C_DIS
LIN {X -0.102,Y -181.256,Z 700.752,A 0.000,B 0.000,C 90.000,E1 135.324} C_DIS
LIN {X 0.028,Y -186.730,Z 700.733,A 0.000,B 0.000,C 90.000,E1 131.919} C_DIS
LIN {X -0.044,Y -191.339,Z 700.719,A 0.000,B 0.000,C 90.000,E1 129.439} C_DIS
LIN {X 0.081,Y -289.525,Z 700.719,A 0.000,B 0.000,C 90.000,E1 129.402} C_DIS
LIN {X 0.019,Y -292.253,Z 700.719,A 0.000,B 0.000,C 90.000,E1 129.358} C_DIS
LIN {X -0.123,Y -295.841,Z 700.718,A 0.000,B 0.000,C 90.000,E1 129.197} C_DIS
LIN {X -0.036,Y -298.058,Z 700.717,A 0.000,B 0.000,C 90.000,E1 128.991} C_DIS
LIN {X -0.093,Y -301.151,Z 700.714,A 0.000,B 0.000,C 90.000,E1 128.624} C_DIS
LIN {X 0.106,Y -303.096,Z 700.713,A 0.000,B 0.000,C 90.000,E1 128.257} C_DIS
LIN {X 0.066,Y -304.610,Z 700.711,A 0.000,B 0.000,C 90.000,E1 127.935} C_DIS
LIN {X 0.081,Y -305.801,Z 700.709,A 0.000,B 0.000,C 90.000,E1 127.604} C_DIS
LIN {X -0.032,Y -316.443,Z 700.689,A 0.000,B 0.000,C 90.000,E1 124.040} C_DIS
LIN {X 0.142,Y -326.464,Z 700.673,A 0.000,B 0.000,C 90.000,E1 121.131} C_DIS
LIN {X -0.181,Y -337.812,Z 700.657,A 0.000,B 0.000,C 90.000,E1 118.359} C_DIS
LIN {X 0.107,Y -350.584,Z 700.642,A 0.000,B 0.000,C 90.000,E1 115.540} C_DIS
LIN {X 0.084,Y -363.228,Z 700.629,A 0.000,B 0.000,C 90.000,E1 113.131} C_DIS
LIN {X -0.062,Y -377.179,Z 700.615,A 0.000,B 0.000,C 90.000,E1 110.791} C_DIS
LIN {X -0.120,Y -392.539,Z 700.603,A 0.000,B 0.000,C 90.000,E1 108.489} C_DIS
LIN {X 0.092,Y -409.418,Z 700.590,A 0.000,B 0.000,C 90.000,E1 106.205} C_DIS
LIN {X 0.106,Y -427.940,Z 700.578,A 0.000,B 0.000,C 90.000,E1 104.008} C_DIS
LIN {X -0.178,Y -447.835,Z 700.566,A 0.000,B 0.000,C 90.000,E1 101.951} C_DIS
LIN {X -0.110,Y -468.325,Z 700.556,A 0.000,B 0.000,C 90.000,E1 100.018} C_DIS
LIN {X -0.147,Y -470.476,Z 700.554,A 0.000,B 0.000,C 90.000,E1 99.792} C_DIS
LIN {X 0.168,Y -472.251,Z 700.553,A 0.000,B 0.000,C 90.000,E1 99.500} C_DIS
LIN {X 0.018,Y -473.584,Z 700.551,A 0.000,B 0.000,C 90.000,E1 99.265} C_DIS
LIN {X 0.131,Y -475.254,Z 700.549,A 0.000,B 0.000,C 90.000,E1 98.746} C_DIS
LIN {X -0.148,Y -475.856,Z 700.546,A 0.000,B 0.000,C 90.000,E1 98.276} C_DIS
LIN {X -0.017,Y -475.493,Z 700.543,A 0.000,B 0.000,C 90.000,E1 97.757} C_DIS
LIN {X 0.119,Y -474.112,Z 700.540,A 0.000,B 0.000,C 90.000,E1 97.239} C_DIS
LIN {X -0.021,Y -472.970,Z 700.539,A 0.000,B 0.000,C 90.000,E1 97.004} C_DIS
LIN {X 0.105,Y -469.738,Z 700.536,A 0.000,B 0.000,C 90.000,E1 96.486} C_DIS
LIN {X 0.163,Y -451.768,Z 700.521,A 0.000,B 0.000,C 90.000,E1 93.669} C_DIS
LIN {X -0.093,Y -437.096,Z 700.506,A 0.000,B 0.000,C 90.000,E1 91.088} C_DIS
LIN {X -0.021,Y -428.119,Z 700.497,A 0.000,B 0.000,C 90.000,E1 89.484} C_DIS
LIN {X 0.008,Y -417.263,Z 700.487,A 0.000,B 0.000,C 90.000,E1 87.593} C_DIS
LIN {X -0.158,Y -406.283,Z 700.476,A 0.000,B 0.000,C 90.000,E1 85.698} C_DIS
LIN {X -0.116,Y -395.327,Z 700.465,A 0.000,B 0.000,C 90.000,E1 83.742} C_DIS
LIN {X -0.155,Y -380.027,Z 700.449,A 0.000,B 0.000,C 90.000,E1 80.905} C_DIS
LIN {X -0.125,Y -368.289,Z 700.436,A 0.000,B 0.000,C 90.000,E1 78.578} C_DIS
LIN {X 0.021,Y -354.111,Z 700.420,A 0.000,B 0.000,C 90.000,E1 75.589} C_DIS
LIN {X 0.082,Y -340.605,Z 700.403,A 0.000,B 0.000,C 90.000,E1 72.543} C_DIS
LIN {X 0.110,Y -330.147,Z 700.389,A 0.000,B 0.000,C 90.000,E1 70.061} C_DIS
LIN {X 0.001,Y -317.940,Z 700.372,A 0.000,B 0.000,C 90.000,E1 66.922} C_DIS
LIN {X 0.010,Y -308.263,Z 700.356,A 0.000,B 0.000,C 90.000,E1 64.024} C_DIS
LIN {X 0.050,Y -298.586,Z 700.338,A 0.000,B 0.000,C 90.000,E1 60.745} C_DIS
LIN {X -0.140,Y -289.542,Z 700.319,A 0.000,B 0.000,C 90.000,E1 57.454} C_DIS
LIN {X 0.175,Y -282.664,Z 700.304,A 0.000,B 0.000,C 90.000,E1 54.689} C_DIS
LIN {X -0.039,Y -277.610,Z 700.293,A 0.000,B 0.000,C 90.000,E1 52.683} C_DIS
LIN {X 0.039,Y -272.426,Z 700.281,A 0.000,B 0.000,C 90.000,E1 50.598} C_DIS
LIN {X -0.053,Y -267.077,Z 700.270,A 0.000,B 0.000,C 90.000,E1 48.528} C_DIS
LIN {X 0.131,Y -261.357,Z 700.258,A 0.000,B 0.000,C 90.000,E1 46.377} C_DIS
LIN {X 0.005,Y -255.459,Z 700.246,A 0.000,B 0.000,C 90.000,E1 44.271} C_DIS
LIN {X -0.045,Y -249.432,Z 700.234,A 0.000,B 0.000,C 90.000,E1 42.123} C_DIS
LIN {X -0.007,Y -243.222,Z 700.222,A 0.000,B 0.000,C 90.000,E1 39.930} C_DIS
LIN {X 0.040,Y -233.161,Z 700.201,A 0.000,B 0.000,C 90.000,E1 36.217} C_DIS
LIN {X -0.068,Y -223.940,Z 700.180,A 0.000,B 0.000,C 90.000,E1 32.467} C_DIS
LIN {X -0.132,Y -217.284,Z 700.163,A 0.000,B 0.000,C 90.000,E1 29.411} C_DIS
LIN {X 0.101,Y -211.495,Z 700.146,A 0.000,B 0.000,C 90.000,E1 26.232} C_DIS
LIN {X 0.096,Y -206.445,Z 700.128,A 0.000,B 0.000,C 90.000,E1 23.078} C_DIS
LIN {X 0.096,Y -201.296,Z 700.106,A 0.000,B 0.000,C 90.000,E1 19.087} C_DIS
LIN {X 0.058,Y -197.323,Z 700.084,A 0.000,B 0.000,C 90.000,E1 15.064} C_DIS
LIN {X 0.001,Y -193.992,Z 700.057,A 0.000,B 0.000,C 90.000,E1 10.197} C_DIS
LIN {X 0.029,Y -191.837,Z 700.016,A 0.000,B 0.000,C 90.000,E1 2.808} C_DIS
LIN {X -0.060,Y -193.651,Z 699.965,A 0.000,B 0.000,C 90.000,E1 353.799} C_DIS
LIN {X 0.018,Y -196.670,Z 699.938,A 0.000,B 0.000,C 90.000,E1 348.870} C_DIS
LIN {X 0.012,Y -200.292,Z 699.916,A 0.000,B 0.000,C 90.000,E1 344.810} C_DIS
LIN {X 0.004,Y -204.884,Z 699.893,A 0.000,B 0.000,C 90.000,E1 340.786} C_DIS
LIN {X 0.028,Y -210.301,Z 699.871,A 0.000,B 0.000,C 90.000,E1 336.794} C_DIS
LIN {X -0.029,Y -216.455,Z 699.849,A 0.000,B 0.000,C 90.000,E1 332.871} C_DIS
LIN {X -0.071,Y -223.332,Z 699.828,A 0.000,B 0.000,C 90.000,E1 328.997} C_DIS
LIN {X -0.128,Y -230.805,Z 699.806,A 0.000,B 0.000,C 90.000,E1 325.182} C_DIS
LIN {X 0.022,Y -238.895,Z 699.785,A 0.000,B 0.000,C 90.000,E1 321.376} C_DIS
LIN {X -0.002,Y -247.917,Z 699.765,A 0.000,B 0.000,C 90.000,E1 317.676} C_DIS
LIN {X 0.060,Y -257.982,Z 699.745,A 0.000,B 0.000,C 90.000,E1 314.028} C_DIS
LIN {X 0.117,Y -269.176,Z 699.725,A 0.000,B 0.000,C 90.000,E1 310.458} C_DIS
LIN {X -0.069,Y -280.362,Z 699.708,A 0.000,B 0.000,C 90.000,E1 307.363} C_DIS
LIN {X 0.162,Y -294.128,Z 699.689,A 0.000,B 0.000,C 90.000,E1 303.913} C_DIS
LIN {X 0.196,Y -309.302,Z 699.670,A 0.000,B 0.000,C 90.000,E1 300.590} C_DIS
LIN {X 0.074,Y -322.593,Z 699.656,A 0.000,B 0.000,C 90.000,E1 298.025} C_DIS
LIN {X -0.066,Y -340.568,Z 699.638,A 0.000,B 0.000,C 90.000,E1 294.899} C_DIS
LIN {X -0.111,Y -357.866,Z 699.623,A 0.000,B 0.000,C 90.000,E1 292.153} C_DIS
LIN {X -0.117,Y -371.938,Z 699.611,A 0.000,B 0.000,C 90.000,E1 290.066} C_DIS
LIN {X -0.072,Y -385.163,Z 699.602,A 0.000,B 0.000,C 90.000,E1 288.308} C_DIS
LIN {X 0.108,Y -399.137,Z 699.592,A 0.000,B 0.000,C 90.000,E1 286.567} C_DIS
LIN {X 0.048,Y -412.984,Z 699.583,A 0.000,B 0.000,C 90.000,E1 284.898} C_DIS
LIN {X -0.023,Y -424.384,Z 699.575,A 0.000,B 0.000,C 90.000,E1 283.536} C_DIS
LIN {X -0.019,Y -435.426,Z 699.568,A 0.000,B 0.000,C 90.000,E1 282.187} C_DIS
LIN {X 0.144,Y -445.772,Z 699.560,A 0.000,B 0.000,C 90.000,E1 280.838} C_DIS
LIN {X 0.041,Y -463.836,Z 699.547,A 0.000,B 0.000,C 90.000,E1 278.511} C_DIS
LIN {X 0.173,Y -471.647,Z 699.542,A 0.000,B 0.000,C 90.000,E1 277.473} C_DIS
LIN {X 0.128,Y -476.881,Z 699.537,A 0.000,B 0.000,C 90.000,E1 276.720} C_DIS
LIN {X 0.129,Y -481.238,Z 699.533,A 0.000,B 0.000,C 90.000,E1 275.967} C_DIS
LIN {X -0.237,Y -483.588,Z 699.530,A 0.000,B 0.000,C 90.000,E1 275.511} C_DIS
LIN {X 0.111,Y -484.594,Z 699.529,A 0.000,B 0.000,C 90.000,E1 275.220} C_DIS
LIN {X -0.190,Y -486.277,Z 699.526,A 0.000,B 0.000,C 90.000,E1 274.759} C_DIS
LIN {X -0.041,Y -487.515,Z 699.524,A 0.000,B 0.000,C 90.000,E1 274.245} C_DIS
LIN {X 0.158,Y -488.357,Z 699.521,A 0.000,B 0.000,C 90.000,E1 273.726} C_DIS
LIN {X -0.156,Y -488.797,Z 699.518,A 0.000,B 0.000,C 90.000,E1 273.269} C_DIS
LIN {X 0.051,Y -488.898,Z 699.515,A 0.000,B 0.000,C 90.000,E1 272.751} C_DIS
LIN {X 0.235,Y -488.684,Z 699.513,A 0.000,B 0.000,C 90.000,E1 272.236} C_DIS
LIN {X -0.050,Y -488.132,Z 699.510,A 0.000,B 0.000,C 90.000,E1 271.776} C_DIS
LIN {X 0.134,Y -487.206,Z 699.507,A 0.000,B 0.000,C 90.000,E1 271.260} C_DIS
LIN {X -0.169,Y -485.862,Z 699.504,A 0.000,B 0.000,C 90.000,E1 270.802} C_DIS
LIN {X 0.009,Y -484.080,Z 699.502,A 0.000,B 0.000,C 90.000,E1 270.286} C_DIS
LIN {X 0.179,Y -481.709,Z 699.499,A 0.000,B 0.000,C 90.000,E1 269.771} C_DIS
LIN {X -0.149,Y -478.695,Z 699.496,A 0.000,B 0.000,C 90.000,E1 269.312} C_DIS
LIN {X -0.013,Y -474.858,Z 699.493,A 0.000,B 0.000,C 90.000,E1 268.797} C_DIS
LIN {X 0.100,Y -470.034,Z 699.491,A 0.000,B 0.000,C 90.000,E1 268.282} C_DIS
LIN {X -0.018,Y -467.273,Z 699.489,A 0.000,B 0.000,C 90.000,E1 268.051} C_DIS
LIN {X -0.016,Y -461.211,Z 699.487,A 0.000,B 0.000,C 90.000,E1 267.593} C_DIS
LIN {X 0.113,Y -457.776,Z 699.485,A 0.000,B 0.000,C 90.000,E1 267.364} C_DIS
LIN {X 0.018,Y -450.816,Z 699.483,A 0.000,B 0.000,C 90.000,E1 267.020} C_DIS
LIN {X 0.019,Y -443.369,Z 699.482,A 0.000,B 0.000,C 90.000,E1 266.731} C_DIS
LIN {X 0.034,Y -439.909,Z 699.481,A 0.000,B 0.000,C 90.000,E1 266.617} C_DIS
LIN {X -0.127,Y -431.549,Z 699.480,A 0.000,B 0.000,C 90.000,E1 266.445} C_DIS
LIN {X 0.195,Y -420.595,Z 699.479,A 0.000,B 0.000,C 90.000,E1 266.274} C_DIS
LIN {X 0.021,Y -414.003,Z 699.479,A 0.000,B 0.000,C 90.000,E1 266.274} C_DIS
LIN {X -0.010,Y -180.933,Z 699.479,A 0.000,B 0.000,C 90.000,E1 266.274} C_DIS
LIN {X 0.034,Y -180.780,Z 699.471,A 0.000,B 0.000,C 90.000,E1 264.723} C_DIS
LIN {X 0.071,Y -178.994,Z 699.444,A 0.000,B 0.000,C 90.000,E1 259.982} C_DIS
LIN {X -0.011,Y -178.576,Z 699.440,A 0.000,B 0.000,C 90.000,E1 259.162} C_DIS
LIN {X 0.052,Y -175.630,Z 699.411,A 0.000,B 0.000,C 90.000,E1 254.047} C_DIS
LIN {X -0.050,Y -172.349,Z 699.388,A 0.000,B 0.000,C 90.000,E1 249.806} C_DIS
LIN {X -0.095,Y -171.131,Z 699.378,A 0.000,B 0.000,C 90.000,E1 248.103} C_DIS
LIN {X -0.050,Y -167.438,Z 699.354,A 0.000,B 0.000,C 90.000,E1 243.768} C_DIS
LIN {X 0.032,Y -166.834,Z 699.349,A 0.000,B 0.000,C 90.000,E1 242.871} C_DIS
LIN {X -0.050,Y -162.817,Z 699.325,A 0.000,B 0.000,C 90.000,E1 238.535} C_DIS
LIN {X 0.014,Y -161.503,Z 699.315,A 0.000,B 0.000,C 90.000,E1 236.755} C_DIS
LIN {X -0.034,Y -157.500,Z 699.291,A 0.000,B 0.000,C 90.000,E1 232.351} C_DIS
LIN {X 0.001,Y -155.520,Z 699.276,A 0.000,B 0.000,C 90.000,E1 229.666} C_DIS
LIN {X 0.051,Y -151.819,Z 699.251,A 0.000,B 0.000,C 90.000,E1 225.162} C_DIS
LIN {X 0.063,Y -150.033,Z 699.236,A 0.000,B 0.000,C 90.000,E1 222.447} C_DIS
LIN {X -0.023,Y -146.852,Z 699.211,A 0.000,B 0.000,C 90.000,E1 217.935} C_DIS
LIN {X -0.005,Y -145.435,Z 699.195,A 0.000,B 0.000,C 90.000,E1 215.185} C_DIS
LIN {X -0.009,Y -142.857,Z 699.170,A 0.000,B 0.000,C 90.000,E1 210.590} C_DIS
LIN {X 0.043,Y -141.472,Z 699.149,A 0.000,B 0.000,C 90.000,E1 206.873} C_DIS
LIN {X 0.034,Y -139.379,Z 699.113,A 0.000,B 0.000,C 90.000,E1 200.375} C_DIS
LIN {X 0.024,Y -138.831,Z 699.098,A 0.000,B 0.000,C 90.000,E1 197.583} C_DIS
LIN {X -0.048,Y -138.354,Z 699.056,A 0.000,B 0.000,C 90.000,E1 190.141} C_DIS
LIN {X -0.053,Y -139.526,Z 699.004,A 0.000,B 0.000,C 90.000,E1 180.802} C_DIS
LIN {X 0.039,Y -141.198,Z 698.973,A 0.000,B 0.000,C 90.000,E1 175.179} C_DIS
LIN {X -0.002,Y -142.574,Z 698.958,A 0.000,B 0.000,C 90.000,E1 172.413} C_DIS
LIN {X -0.047,Y -144.865,Z 698.932,A 0.000,B 0.000,C 90.000,E1 167.813} C_DIS
LIN {X 0.050,Y -147.490,Z 698.912,A 0.000,B 0.000,C 90.000,E1 164.102} C_DIS
LIN {X -0.017,Y -150.079,Z 698.891,A 0.000,B 0.000,C 90.000,E1 160.477} C_DIS
LIN {X -0.003,Y -153.429,Z 698.871,A 0.000,B 0.000,C 90.000,E1 156.847} C_DIS
LIN {X -0.016,Y -156.849,Z 698.851,A 0.000,B 0.000,C 90.000,E1 153.256} C_DIS
LIN {X 0.056,Y -160.931,Z 698.832,A 0.000,B 0.000,C 90.000,E1 149.665} C_DIS
LIN {X 0.000,Y -163.055,Z 698.822,A 0.000,B 0.000,C 90.000,E1 147.916} C_DIS
LIN {X 0.004,Y -167.450,Z 698.802,A 0.000,B 0.000,C 90.000,E1 144.402} C_DIS
LIN {X -0.086,Y -171.287,Z 698.788,A 0.000,B 0.000,C 90.000,E1 141.823} C_DIS
LIN {X 0.083,Y -176.181,Z 698.769,A 0.000,B 0.000,C 90.000,E1 138.324} C_DIS
LIN {X -0.051,Y -180.455,Z 698.754,A 0.000,B 0.000,C 90.000,E1 135.810} C_DIS
LIN {X -0.076,Y -185.859,Z 698.736,A 0.000,B 0.000,C 90.000,E1 132.447} C_DIS
LIN {X -0.029,Y -191.332,Z 698.719,A 0.000,B 0.000,C 90.000,E1 129.439} C_DIS
LIN {X -0.075,Y -289.694,Z 698.719,A 0.000,B 0.000,C 90.000,E1 129.439} C_DIS
LIN {X -0.121,Y -294.678,Z 698.718,A 0.000,B 0.000,C 90.000,E1 129.277} C_DIS
LIN {X -0.106,Y -296.880,Z 698.717,A 0.000,B 0.000,C 90.000,E1 129.116} C_DIS
LIN {X -0.021,Y -300.756,Z 698.715,A 0.000,B 0.000,C 90.000,E1 128.669} C_DIS
LIN {X -0.134,Y -302.668,Z 698.713,A 0.000,B 0.000,C 90.000,E1 128.382} C_DIS
LIN {X -0.008,Y -304.171,Z 698.711,A 0.000,B 0.000,C 90.000,E1 128.051} C_DIS
LIN {X -0.048,Y -305.448,Z 698.710,A 0.000,B 0.000,C 90.000,E1 127.729} C_DIS
LIN {X 0.136,Y -317.150,Z 698.688,A 0.000,B 0.000,C 90.000,E1 123.785} C_DIS
LIN {X 0.060,Y -327.272,Z 698.672,A 0.000,B 0.000,C 90.000,E1 120.924} C_DIS
LIN {X 0.056,Y -338.724,Z 698.656,A 0.000,B 0.000,C 90.000,E1 118.103} C_DIS
LIN {X 0.059,Y -351.614,Z 698.641,A 0.000,B 0.000,C 90.000,E1 115.335} C_DIS
LIN {X -0.091,Y -364.368,Z 698.627,A 0.000,B 0.000,C 90.000,E1 112.950} C_DIS
LIN {X 0.143,Y -378.438,Z 698.614,A 0.000,B 0.000,C 90.000,E1 110.556} C_DIS
LIN {X -0.120,Y -393.925,Z 698.602,A 0.000,B 0.000,C 90.000,E1 108.290} C_DIS
LIN {X -0.001,Y -410.943,Z 698.589,A 0.000,B 0.000,C 90.000,E1 106.024} C_DIS
LIN {X 0.043,Y -429.614,Z 698.577,A 0.000,B 0.000,C 90.000,E1 103.828} C_DIS
LIN {X -0.149,Y -449.593,Z 698.565,A 0.000,B 0.000,C 90.000,E1 101.771} C_DIS
LIN {X -0.007,Y -467.524,Z 698.556,A 0.000,B 0.000,C 90.000,E1 100.074} C_DIS
LIN {X -0.051,Y -469.891,Z 698.555,A 0.000,B 0.000,C 90.000,E1 99.849} C_DIS
LIN {X -0.120,Y -471.764,Z 698.553,A 0.000,B 0.000,C 90.000,E1 99.613} C_DIS
LIN {X -0.191,Y -473.184,Z 698.552,A 0.000,B 0.000,C 90.000,E1 99.378} C_DIS
LIN {X -0.084,Y -475.081,Z 698.549,A 0.000,B 0.000,C 90.000,E1 98.859} C_DIS
LIN {X 0.037,Y -475.871,Z 698.546,A 0.000,B 0.000,C 90.000,E1 98.341} C_DIS
LIN {X 0.234,Y -475.687,Z 698.544,A 0.000,B 0.000,C 90.000,E1 97.814} C_DIS
LIN {X -0.101,Y -474.508,Z 698.541,A 0.000,B 0.000,C 90.000,E1 97.352} C_DIS
LIN {X 0.172,Y -473.489,Z 698.539,A 0.000,B 0.000,C 90.000,E1 97.068} C_DIS
LIN {X 0.034,Y -472.120,Z 698.538,A 0.000,B 0.000,C 90.000,E1 96.834} C_DIS
LIN {X -0.029,Y -452.373,Z 698.521,A 0.000,B 0.000,C 90.000,E1 93.784} C_DIS
LIN {X 0.173,Y -437.680,Z 698.506,A 0.000,B 0.000,C 90.000,E1 91.146} C_DIS
LIN {X -0.180,Y -428.733,Z 698.498,A 0.000,B 0.000,C 90.000,E1 89.599} C_DIS
LIN {X 0.178,Y -419.483,Z 698.489,A 0.000,B 0.000,C 90.000,E1 87.936} C_DIS
LIN {X 0.024,Y -408.501,Z 698.478,A 0.000,B 0.000,C 90.000,E1 86.045} C_DIS
LIN {X 0.104,Y -397.556,Z 698.467,A 0.000,B 0.000,C 90.000,E1 84.090} C_DIS
LIN {X 0.116,Y -382.165,Z 698.451,A 0.000,B 0.000,C 90.000,E1 81.254} C_DIS
LIN {X 0.190,Y -370.399,Z 698.439,A 0.000,B 0.000,C 90.000,E1 78.926} C_DIS
LIN {X -0.002,Y -354.765,Z 698.421,A 0.000,B 0.000,C 90.000,E1 75.700} C_DIS
LIN {X -0.007,Y -339.918,Z 698.402,A 0.000,B 0.000,C 90.000,E1 72.362} C_DIS
LIN {X 0.008,Y -329.516,Z 698.388,A 0.000,B 0.000,C 90.000,E1 69.880} C_DIS
LIN {X -0.057,Y -316.307,Z 698.369,A 0.000,B 0.000,C 90.000,E1 66.410} C_DIS
LIN {X -0.135,Y -304.887,Z 698.349,A 0.000,B 0.000,C 90.000,E1 62.871} C_DIS
LIN {X 0.091,Y -295.476,Z 698.331,A 0.000,B 0.000,C 90.000,E1 59.537} C_DIS
LIN {X -0.033,Y -286.688,Z 698.312,A 0.000,B 0.000,C 90.000,E1 56.215} C_DIS
LIN {X -0.025,Y -279.906,Z 698.297,A 0.000,B 0.000,C 90.000,E1 53.497} C_DIS
LIN {X -0.119,Y -274.799,Z 698.286,A 0.000,B 0.000,C 90.000,E1 51.457} C_DIS
LIN {X -0.133,Y -269.538,Z 698.274,A 0.000,B 0.000,C 90.000,E1 49.380} C_DIS
LIN {X 0.101,Y -263.967,Z 698.263,A 0.000,B 0.000,C 90.000,E1 47.229} C_DIS
LIN {X 0.028,Y -258.106,Z 698.251,A 0.000,B 0.000,C 90.000,E1 45.121} C_DIS
LIN {X 0.023,Y -252.114,Z 698.239,A 0.000,B 0.000,C 90.000,E1 42.975} C_DIS
LIN {X -0.077,Y -245.968,Z 698.227,A 0.000,B 0.000,C 90.000,E1 40.825} C_DIS
LIN {X -0.128,Y -235.733,Z 698.206,A 0.000,B 0.000,C 90.000,E1 37.156} C_DIS
LIN {X -0.019,Y -226.258,Z 698.185,A 0.000,B 0.000,C 90.000,E1 33.372} C_DIS
LIN {X -0.101,Y -219.361,Z 698.168,A 0.000,B 0.000,C 90.000,E1 30.335} C_DIS
LIN {X -0.002,Y -213.311,Z 698.151,A 0.000,B 0.000,C 90.000,E1 27.206} C_DIS
LIN {X -0.058,Y -208.020,Z 698.134,A 0.000,B 0.000,C 90.000,E1 24.079} C_DIS
LIN {X 0.069,Y -202.614,Z 698.112,A 0.000,B 0.000,C 90.000,E1 20.066} C_DIS
LIN {X -0.054,Y -198.340,Z 698.089,A 0.000,B 0.000,C 90.000,E1 16.079} C_DIS
LIN {X 0.012,Y -194.702,Z 698.062,A 0.000,B 0.000,C 90.000,E1 11.186} C_DIS
LIN {X -0.017,Y -192.193,Z 698.026,A 0.000,B 0.000,C 90.000,E1 4.645} C_DIS
LIN {X -0.055,Y -193.764,Z 697.965,A 0.000,B 0.000,C 90.000,E1 353.799} C_DIS
LIN {X 0.027,Y -196.779,Z 697.938,A 0.000,B 0.000,C 90.000,E1 348.870} C_DIS
LIN {X 0.026,Y -200.375,Z 697.916,A 0.000,B 0.000,C 90.000,E1 344.810} C_DIS
LIN {X 0.020,Y -204.962,Z 697.893,A 0.000,B 0.000,C 90.000,E1 340.786} C_DIS
LIN {X 0.046,Y -210.368,Z 697.871,A 0.000,B 0.000,C 90.000,E1 336.794} C_DIS
LIN {X -0.007,Y -216.502,Z 697.849,A 0.000,B 0.000,C 90.000,E1 332.871} C_DIS
LIN {X -0.049,Y -223.372,Z 697.828,A 0.000,B 0.000,C 90.000,E1 328.997} C_DIS
LIN {X -0.102,Y -230.842,Z 697.806,A 0.000,B 0.000,C 90.000,E1 325.182} C_DIS
LIN {X 0.050,Y -238.917,Z 697.785,A 0.000,B 0.000,C 90.000,E1 321.376} C_DIS
LIN {X 0.027,Y -247.939,Z 697.765,A 0.000,B 0.000,C 90.000,E1 317.676} C_DIS
LIN {X 0.090,Y -257.985,Z 697.745,A 0.000,B 0.000,C 90.000,E1 314.028} C_DIS
LIN {X 0.149,Y -269.184,Z 697.725,A 0.000,B 0.000,C 90.000,E1 310.458} C_DIS
LIN {X -0.034,Y -280.368,Z 697.708,A 0.000,B 0.000,C 90.000,E1 307.363} C_DIS
LIN {X 0.197,Y -294.117,Z 697.689,A 0.000,B 0.000,C 90.000,E1 303.913} C_DIS
LIN {X -0.190,Y -309.308,Z 697.670,A 0.000,B 0.000,C 90.000,E1 300.669} C_DIS
LIN {X 0.034,Y -320.854,Z 697.658,A 0.000,B 0.000,C 90.000,E1 298.359} C_DIS
LIN {X -0.105,Y -334.960,Z 697.643,A 0.000,B 0.000,C 90.000,E1 295.848} C_DIS
LIN {X 0.130,Y -349.971,Z 697.630,A 0.000,B 0.000,C 90.000,E1 293.334} C_DIS
LIN {X 0.158,Y -365.671,Z 697.616,A 0.000,B 0.000,C 90.000,E1 290.918} C_DIS
LIN {X 0.113,Y -376.084,Z 697.608,A 0.000,B 0.000,C 90.000,E1 289.450} C_DIS
LIN {X 0.088,Y -396.637,Z 697.594,A 0.000,B 0.000,C 90.000,E1 286.858} C_DIS
LIN {X -0.021,Y -410.522,Z 697.584,A 0.000,B 0.000,C 90.000,E1 285.190} C_DIS
LIN {X 0.012,Y -424.205,Z 697.575,A 0.000,B 0.000,C 90.000,E1 283.536} C_DIS
LIN {X 0.014,Y -435.225,Z 697.568,A 0.000,B 0.000,C 90.000,E1 282.187} C_DIS
LIN {X 0.175,Y -445.542,Z 697.560,A 0.000,B 0.000,C 90.000,E1 280.838} C_DIS
LIN {X 0.066,Y -463.609,Z 697.547,A 0.000,B 0.000,C 90.000,E1 278.511} C_DIS
LIN {X 0.198,Y -471.449,Z 697.542,A 0.000,B 0.000,C 90.000,E1 277.473} C_DIS
LIN {X 0.152,Y -476.676,Z 697.537,A 0.000,B 0.000,C 90.000,E1 276.720} C_DIS
LIN {X -0.190,Y -479.711,Z 697.535,A 0.000,B 0.000,C 90.000,E1 276.258} C_DIS
LIN {X -0.038,Y -482.264,Z 697.532,A 0.000,B 0.000,C 90.000,E1 275.739} C_DIS
LIN {X 0.131,Y -484.438,Z 697.529,A 0.000,B 0.000,C 90.000,E1 275.220} C_DIS
LIN {X -0.170,Y -486.096,Z 697.526,A 0.000,B 0.000,C 90.000,E1 274.759} C_DIS
LIN {X -0.021,Y -487.379,Z 697.524,A 0.000,B 0.000,C 90.000,E1 274.245} C_DIS
LIN {X 0.175,Y -488.215,Z 697.521,A 0.000,B 0.000,C 90.000,E1 273.726} C_DIS
LIN {X -0.139,Y -488.674,Z 697.518,A 0.000,B 0.000,C 90.000,E1 273.269} C_DIS
LIN {X 0.066,Y -488.767,Z 697.515,A 0.000,B 0.000,C 90.000,E1 272.751} C_DIS
LIN {X -0.238,Y -488.565,Z 697.513,A 0.000,B 0.000,C 90.000,E1 272.293} C_DIS
LIN {X -0.035,Y -488.041,Z 697.510,A 0.000,B 0.000,C 90.000,E1 271.776} C_DIS
LIN {X 0.148,Y -487.110,Z 697.507,A 0.000,B 0.000,C 90.000,E1 271.260} C_DIS
LIN {X -0.156,Y -485.801,Z 697.504,A 0.000,B 0.000,C 90.000,E1 270.802} C_DIS
LIN {X 0.022,Y -484.033,Z 697.502,A 0.000,B 0.000,C 90.000,E1 270.286} C_DIS
LIN {X 0.191,Y -481.662,Z 697.499,A 0.000,B 0.000,C 90.000,E1 269.771} C_DIS
LIN {X -0.138,Y -478.644,Z 697.496,A 0.000,B 0.000,C 90.000,E1 269.312} C_DIS
LIN {X -0.002,Y -474.869,Z 697.493,A 0.000,B 0.000,C 90.000,E1 268.797} C_DIS
LIN {X -0.180,Y -472.618,Z 697.492,A 0.000,B 0.000,C 90.000,E1 268.568} C_DIS
LIN {X -0.001,Y -467.350,Z 697.489,A 0.000,B 0.000,C 90.000,E1 268.051} C_DIS
LIN {X 0.000,Y -461.266,Z 697.487,A 0.000,B 0.000,C 90.000,E1 267.593} C_DIS
LIN {X 0.079,Y -454.628,Z 697.484,A 0.000,B 0.000,C 90.000,E1 267.192} C_DIS
LIN {X -0.181,Y -447.455,Z 697.483,A 0.000,B 0.000,C 90.000,E1 266.906} C_DIS
LIN {X 0.070,Y -440.174,Z 697.481,A 0.000,B 0.000,C 90.000,E1 266.617} C_DIS
LIN {X -0.125,Y -431.833,Z 697.480,A 0.000,B 0.000,C 90.000,E1 266.445} C_DIS
LIN {X 0.208,Y -421.453,Z 697.479,A 0.000,B 0.000,C 90.000,E1 266.274} C_DIS
LIN {X -0.034,Y -413.191,Z 697.479,A 0.000,B 0.000,C 90.000,E1 266.274} C_DIS
LIN {X -0.036,Y -180.933,Z 697.479,A 0.000,B 0.000,C 90.000,E1 266.274} C_DIS
LIN {X 0.023,Y -180.779,Z 697.471,A 0.000,B 0.000,C 90.000,E1 264.723} C_DIS
LIN {X 0.060,Y -178.993,Z 697.444,A 0.000,B 0.000,C 90.000,E1 259.982} C_DIS
LIN {X -0.022,Y -178.574,Z 697.440,A 0.000,B 0.000,C 90.000,E1 259.162} C_DIS
LIN {X 0.041,Y -175.627,Z 697.411,A 0.000,B 0.000,C 90.000,E1 254.047} C_DIS
LIN {X 0.100,Y -172.347,Z 697.388,A 0.000,B 0.000,C 90.000,E1 249.752} C_DIS
LIN {X 0.053,Y -171.126,Z 697.378,A 0.000,B 0.000,C 90.000,E1 248.050} C_DIS
LIN {X -0.061,Y -167.436,Z 697.354,A 0.000,B 0.000,C 90.000,E1 243.768} C_DIS
LIN {X 0.022,Y -166.831,Z 697.349,A 0.000,B 0.000,C 90.000,E1 242.871} C_DIS
LIN {X -0.060,Y -162.813,Z 697.325,A 0.000,B 0.000,C 90.000,E1 238.535} C_DIS
LIN {X 0.003,Y -161.500,Z 697.315,A 0.000,B 0.000,C 90.000,E1 236.755} C_DIS
LIN {X -0.043,Y -157.497,Z 697.291,A 0.000,B 0.000,C 90.000,E1 232.351} C_DIS
LIN {X -0.009,Y -155.517,Z 697.276,A 0.000,B 0.000,C 90.000,E1 229.666} C_DIS
LIN {X 0.041,Y -151.817,Z 697.251,A 0.000,B 0.000,C 90.000,E1 225.162} C_DIS
LIN {X 0.054,Y -150.030,Z 697.236,A 0.000,B 0.000,C 90.000,E1 222.447} C_DIS
LIN {X -0.033,Y -146.849,Z 697.211,A 0.000,B 0.000,C 90.000,E1 217.935} C_DIS
LIN {X -0.014,Y -145.432,Z 697.195,A 0.000,B 0.000,C 90.000,E1 215.185} C_DIS
LIN {X -0.019,Y -142.856,Z 697.170,A 0.000,B 0.000,C 90.000,E1 210.590} C_DIS
LIN {X 0.034,Y -141.471,Z 697.149,A 0.000,B 0.000,C 90.000,E1 206.873} C_DIS
LIN {X 0.024,Y -139.379,Z 697.113,A 0.000,B 0.000,C 90.000,E1 200.375} C_DIS
LIN {X 0.015,Y -138.831,Z 697.098,A 0.000,B 0.000,C 90.000,E1 197.583} C_DIS
LIN {X -0.057,Y -138.353,Z 697.056,A 0.000,B 0.000,C 90.000,E1 190.141} C_DIS
LIN {X -0.062,Y -139.527,Z 697.004,A 0.000,B 0.000,C 90.000,E1 180.802} C_DIS
LIN {X 0.030,Y -141.199,Z 696.973,A 0.000,B 0.000,C 90.000,E1 175.179} C_DIS
LIN {X -0.010,Y -142.576,Z 696.958,A 0.000,B 0.000,C 90.000,E1 172.413} C_DIS
LIN {X -0.056,Y -144.866,Z 696.932,A 0.000,B 0.000,C 90.000,E1 167.813} C_DIS
LIN {X 0.040,Y -147.493,Z 696.912,A 0.000,B 0.000,C 90.000,E1 164.102} C_DIS
LIN {X -0.026,Y -150.082,Z 696.891,A 0.000,B 0.000,C 90.000,E1 160.477} C_DIS
LIN {X -0.013,Y -153.433,Z 696.871,A 0.000,B 0.000,C 90.000,E1 156.847} C_DIS
LIN {X -0.025,Y -156.853,Z 696.851,A 0.000,B 0.000,C 90.000,E1 153.256} C_DIS
LIN {X 0.045,Y -160.936,Z 696.832,A 0.000,B 0.000,C 90.000,E1 149.665} C_DIS
LIN {X -0.010,Y -163.059,Z 696.822,A 0.000,B 0.000,C 90.000,E1 147.916} C_DIS
LIN {X -0.006,Y -167.454,Z 696.802,A 0.000,B 0.000,C 90.000,E1 144.402} C_DIS
LIN {X 0.037,Y -171.292,Z 696.788,A 0.000,B 0.000,C 90.000,E1 141.778} C_DIS
LIN {X 0.073,Y -176.186,Z 696.769,A 0.000,B 0.000,C 90.000,E1 138.324} C_DIS
LIN {X -0.062,Y -180.461,Z 696.754,A 0.000,B 0.000,C 90.000,E1 135.810} C_DIS
LIN {X -0.087,Y -185.865,Z 696.736,A 0.000,B 0.000,C 90.000,E1 132.447} C_DIS
LIN {X 0.020,Y -191.308,Z 696.719,A 0.000,B 0.000,C 90.000,E1 129.439} C_DIS
LIN {X 0.000,Y -288.904,Z 696.719,A 0.000,B 0.000,C 90.000,E1 129.439} C_DIS
LIN {X 0.034,Y -291.152,Z 696.719,A 0.000,B 0.000,C 90.000,E1 129.402} C_DIS
LIN {X -0.124,Y -296.993,Z 696.717,A 0.000,B 0.000,C 90.000,E1 129.116} C_DIS
LIN {X 0.045,Y -300.098,Z 696.715,A 0.000,B 0.000,C 90.000,E1 128.749} C_DIS
LIN {X -0.028,Y -302.107,Z 696.714,A 0.000,B 0.000,C 90.000,E1 128.463} C_DIS
LIN {X -0.101,Y -303.682,Z 696.712,A 0.000,B 0.000,C 90.000,E1 128.177} C_DIS
LIN {X 0.097,Y -305.053,Z 696.710,A 0.000,B 0.000,C 90.000,E1 127.810} C_DIS
LIN {X -0.133,Y -306.132,Z 696.708,A 0.000,B 0.000,C 90.000,E1 127.523} C_DIS
LIN {X -0.048,Y -315.746,Z 696.690,A 0.000,B 0.000,C 90.000,E1 124.246} C_DIS
LIN {X 0.105,Y -325.677,Z 696.674,A 0.000,B 0.000,C 90.000,E1 121.337} C_DIS
LIN {X -0.076,Y -336.928,Z 696.658,A 0.000,B 0.000,C 90.000,E1 118.537} C_DIS
LIN {X 0.180,Y -349.596,Z 696.643,A 0.000,B 0.000,C 90.000,E1 115.720} C_DIS
LIN {X -0.014,Y -362.141,Z 696.630,A 0.000,B 0.000,C 90.000,E1 113.334} C_DIS
LIN {X -0.045,Y -375.985,Z 696.616,A 0.000,B 0.000,C 90.000,E1 110.972} C_DIS
LIN {X -0.134,Y -391.230,Z 696.604,A 0.000,B 0.000,C 90.000,E1 108.671} C_DIS
LIN {X 0.044,Y -407.985,Z 696.591,A 0.000,B 0.000,C 90.000,E1 106.386} C_DIS
LIN {X 0.023,Y -426.373,Z 696.579,A 0.000,B 0.000,C 90.000,E1 104.189} C_DIS
LIN {X 0.173,Y -446.204,Z 696.567,A 0.000,B 0.000,C 90.000,E1 102.063} C_DIS
LIN {X 0.094,Y -469.186,Z 696.555,A 0.000,B 0.000,C 90.000,E1 99.905} C_DIS
LIN {X 0.101,Y -471.181,Z 696.554,A 0.000,B 0.000,C 90.000,E1 99.670} C_DIS
LIN {X 0.029,Y -472.701,Z 696.552,A 0.000,B 0.000,C 90.000,E1 99.443} C_DIS
LIN {X -0.114,Y -473.943,Z 696.551,A 0.000,B 0.000,C 90.000,E1 99.208} C_DIS
LIN {X 0.210,Y -474.854,Z 696.550,A 0.000,B 0.000,C 90.000,E1 98.916} C_DIS
LIN {X -0.136,Y -475.844,Z 696.547,A 0.000,B 0.000,C 90.000,E1 98.454} C_DIS
LIN {X -0.005,Y -475.849,Z 696.544,A 0.000,B 0.000,C 90.000,E1 97.936} C_DIS
LIN {X 0.194,Y -474.876,Z 696.541,A 0.000,B 0.000,C 90.000,E1 97.409} C_DIS
LIN {X -0.141,Y -472.758,Z 696.539,A 0.000,B 0.000,C 90.000,E1 96.947} C_DIS
LIN {X 0.020,Y -457.811,Z 696.526,A 0.000,B 0.000,C 90.000,E1 94.645} C_DIS
LIN {X -0.009,Y -445.521,Z 696.514,A 0.000,B 0.000,C 90.000,E1 92.579} C_DIS
LIN {X -0.049,Y -435.375,Z 696.504,A 0.000,B 0.000,C 90.000,E1 90.745} C_DIS
LIN {X -0.008,Y -426.360,Z 696.495,A 0.000,B 0.000,C 90.000,E1 89.141} C_DIS
LIN {X -0.017,Y -415.471,Z 696.485,A 0.000,B 0.000,C 90.000,E1 87.249} C_DIS
LIN {X 0.180,Y -404.480,Z 696.474,A 0.000,B 0.000,C 90.000,E1 85.298} C_DIS
LIN {X -0.180,Y -393.548,Z 696.463,A 0.000,B 0.000,C 90.000,E1 83.394} C_DIS
LIN {X 0.111,Y -378.388,Z 696.447,A 0.000,B 0.000,C 90.000,E1 80.500} C_DIS
LIN {X 0.076,Y -365.276,Z 696.433,A 0.000,B 0.000,C 90.000,E1 77.881} C_DIS
LIN {X -0.141,Y -351.266,Z 696.416,A 0.000,B 0.000,C 90.000,E1 74.936} C_DIS
LIN {X -0.057,Y -339.273,Z 696.401,A 0.000,B 0.000,C 90.000,E1 72.181} C_DIS
LIN {X -0.083,Y -327.673,Z 696.385,A 0.000,B 0.000,C 90.000,E1 69.390} C_DIS
LIN {X -0.137,Y -315.850,Z 696.368,A 0.000,B 0.000,C 90.000,E1 66.230} C_DIS
LIN {X 0.073,Y -303.571,Z 696.346,A 0.000,B 0.000,C 90.000,E1 62.308} C_DIS
LIN {X 0.134,Y -294.272,Z 696.328,A 0.000,B 0.000,C 90.000,E1 58.997} C_DIS
LIN {X -0.027,Y -285.592,Z 696.309,A 0.000,B 0.000,C 90.000,E1 55.674} C_DIS
LIN {X 0.113,Y -278.876,Z 696.294,A 0.000,B 0.000,C 90.000,E1 52.924} C_DIS
LIN {X -0.003,Y -273.712,Z 696.283,A 0.000,B 0.000,C 90.000,E1 50.884} C_DIS
LIN {X 0.132,Y -268.399,Z 696.271,A 0.000,B 0.000,C 90.000,E1 48.771} C_DIS
LIN {X -0.036,Y -262.725,Z 696.259,A 0.000,B 0.000,C 90.000,E1 46.701} C_DIS
LIN {X -0.133,Y -256.809,Z 696.248,A 0.000,B 0.000,C 90.000,E1 44.595} C_DIS
LIN {X 0.032,Y -250.779,Z 696.236,A 0.000,B 0.000,C 90.000,E1 42.405} C_DIS
LIN {X -0.085,Y -244.559,Z 696.224,A 0.000,B 0.000,C 90.000,E1 40.253} C_DIS
LIN {X 0.016,Y -234.397,Z 696.203,A 0.000,B 0.000,C 90.000,E1 36.537} C_DIS
LIN {X 0.081,Y -224.986,Z 696.182,A 0.000,B 0.000,C 90.000,E1 32.752} C_DIS
LIN {X -0.040,Y -218.262,Z 696.165,A 0.000,B 0.000,C 90.000,E1 29.716} C_DIS
LIN {X -0.075,Y -212.368,Z 696.148,A 0.000,B 0.000,C 90.000,E1 26.616} C_DIS
LIN {X -0.053,Y -207.258,Z 696.130,A 0.000,B 0.000,C 90.000,E1 23.462} C_DIS
LIN {X 0.051,Y -202.027,Z 696.108,A 0.000,B 0.000,C 90.000,E1 19.450} C_DIS
LIN {X 0.037,Y -197.943,Z 696.086,A 0.000,B 0.000,C 90.000,E1 15.426} C_DIS
LIN {X 0.047,Y -194.504,Z 696.059,A 0.000,B 0.000,C 90.000,E1 10.546} C_DIS
LIN {X -0.086,Y -192.128,Z 696.018,A 0.000,B 0.000,C 90.000,E1 3.212} C_DIS
LIN {X -0.050,Y -193.875,Z 695.965,A 0.000,B 0.000,C 90.000,E1 353.799} C_DIS
LIN {X 0.037,Y -196.885,Z 695.938,A 0.000,B 0.000,C 90.000,E1 348.870} C_DIS
LIN {X 0.039,Y -200.461,Z 695.916,A 0.000,B 0.000,C 90.000,E1 344.810} C_DIS
LIN {X 0.036,Y -205.041,Z 695.893,A 0.000,B 0.000,C 90.000,E1 340.786} C_DIS
LIN {X 0.065,Y -210.434,Z 695.871,A 0.000,B 0.000,C 90.000,E1 336.794} C_DIS
LIN {X 0.013,Y -216.550,Z 695.849,A 0.000,B 0.000,C 90.000,E1 332.871} C_DIS
LIN {X -0.025,Y -223.401,Z 695.828,A 0.000,B 0.000,C 90.000,E1 328.997} C_DIS
LIN {X -0.077,Y -230.878,Z 695.806,A 0.000,B 0.000,C 90.000,E1 325.182} C_DIS
LIN {X 0.077,Y -238.946,Z 695.786,A 0.000,B 0.000,C 90.000,E1 321.376} C_DIS
LIN {X -0.111,Y -247.951,Z 695.765,A 0.000,B 0.000,C 90.000,E1 317.715} C_DIS
LIN {X 0.121,Y -257.983,Z 695.745,A 0.000,B 0.000,C 90.000,E1 314.028} C_DIS
LIN {X -0.060,Y -267.993,Z 695.727,A 0.000,B 0.000,C 90.000,E1 310.862} C_DIS
LIN {X -0.109,Y -279.062,Z 695.709,A 0.000,B 0.000,C 90.000,E1 307.729} C_DIS
LIN {X 0.080,Y -292.671,Z 695.690,A 0.000,B 0.000,C 90.000,E1 304.278} C_DIS
LIN {X -0.190,Y -307.739,Z 695.672,A 0.000,B 0.000,C 90.000,E1 301.003} C_DIS
LIN {X 0.072,Y -320.861,Z 695.658,A 0.000,B 0.000,C 90.000,E1 298.359} C_DIS
LIN {X -0.065,Y -334.951,Z 695.644,A 0.000,B 0.000,C 90.000,E1 295.848} C_DIS
LIN {X -0.150,Y -349.904,Z 695.630,A 0.000,B 0.000,C 90.000,E1 293.387} C_DIS
LIN {X -0.143,Y -365.571,Z 695.616,A 0.000,B 0.000,C 90.000,E1 290.972} C_DIS
LIN {X -0.226,Y -378.121,Z 695.607,A 0.000,B 0.000,C 90.000,E1 289.214} C_DIS
LIN {X 0.125,Y -396.467,Z 695.594,A 0.000,B 0.000,C 90.000,E1 286.858} C_DIS
LIN {X 0.014,Y -410.381,Z 695.584,A 0.000,B 0.000,C 90.000,E1 285.190} C_DIS
LIN {X 0.045,Y -424.051,Z 695.575,A 0.000,B 0.000,C 90.000,E1 283.536} C_DIS
LIN {X 0.046,Y -435.002,Z 695.568,A 0.000,B 0.000,C 90.000,E1 282.187} C_DIS
LIN {X -0.011,Y -443.310,Z 695.562,A 0.000,B 0.000,C 90.000,E1 281.130} C_DIS
LIN {X 0.067,Y -459.337,Z 695.550,A 0.000,B 0.000,C 90.000,E1 279.029} C_DIS
LIN {X -0.025,Y -469.361,Z 695.543,A 0.000,B 0.000,C 90.000,E1 277.757} C_DIS
LIN {X -0.090,Y -474.837,Z 695.539,A 0.000,B 0.000,C 90.000,E1 277.004} C_DIS
LIN {X 0.029,Y -478.099,Z 695.536,A 0.000,B 0.000,C 90.000,E1 276.486} C_DIS
LIN {X 0.170,Y -480.904,Z 695.533,A 0.000,B 0.000,C 90.000,E1 275.967} C_DIS
LIN {X -0.198,Y -483.253,Z 695.530,A 0.000,B 0.000,C 90.000,E1 275.511} C_DIS
LIN {X 0.150,Y -484.258,Z 695.529,A 0.000,B 0.000,C 90.000,E1 275.220} C_DIS
LIN {X -0.153,Y -485.957,Z 695.526,A 0.000,B 0.000,C 90.000,E1 274.759} C_DIS
LIN {X -0.005,Y -487.206,Z 695.524,A 0.000,B 0.000,C 90.000,E1 274.245} C_DIS
LIN {X 0.191,Y -488.064,Z 695.521,A 0.000,B 0.000,C 90.000,E1 273.726} C_DIS
LIN {X -0.125,Y -488.528,Z 695.518,A 0.000,B 0.000,C 90.000,E1 273.269} C_DIS
LIN {X 0.080,Y -488.630,Z 695.515,A 0.000,B 0.000,C 90.000,E1 272.751} C_DIS
LIN {X -0.224,Y -488.433,Z 695.513,A 0.000,B 0.000,C 90.000,E1 272.293} C_DIS
LIN {X -0.023,Y -487.918,Z 695.510,A 0.000,B 0.000,C 90.000,E1 271.776} C_DIS
LIN {X 0.160,Y -487.025,Z 695.507,A 0.000,B 0.000,C 90.000,E1 271.260} C_DIS
LIN {X -0.145,Y -485.762,Z 695.504,A 0.000,B 0.000,C 90.000,E1 270.802} C_DIS
LIN {X 0.032,Y -483.989,Z 695.502,A 0.000,B 0.000,C 90.000,E1 270.286} C_DIS
LIN {X 0.201,Y -481.651,Z 695.499,A 0.000,B 0.000,C 90.000,E1 269.771} C_DIS
LIN {X -0.128,Y -478.657,Z 695.496,A 0.000,B 0.000,C 90.000,E1 269.312} C_DIS
LIN {X 0.008,Y -474.869,Z 695.493,A 0.000,B 0.000,C 90.000,E1 268.797} C_DIS
LIN {X -0.171,Y -472.659,Z 695.492,A 0.000,B 0.000,C 90.000,E1 268.568} C_DIS
LIN {X 0.012,Y -467.391,Z 695.489,A 0.000,B 0.000,C 90.000,E1 268.051} C_DIS
LIN {X -0.111,Y -464.359,Z 695.488,A 0.000,B 0.000,C 90.000,E1 267.822} C_DIS
LIN {X -0.001,Y -461.303,Z 695.487,A 0.000,B 0.000,C 90.000,E1 267.593} C_DIS
LIN {X 0.068,Y -454.627,Z 695.484,A 0.000,B 0.000,C 90.000,E1 267.192} C_DIS
LIN {X -0.184,Y -447.534,Z 695.483,A 0.000,B 0.000,C 90.000,E1 266.906} C_DIS
LIN {X 0.059,Y -440.201,Z 695.481,A 0.000,B 0.000,C 90.000,E1 266.617} C_DIS
LIN {X 0.045,Y -435.898,Z 695.481,A 0.000,B 0.000,C 90.000,E1 266.502} C_DIS
LIN {X -0.163,Y -431.767,Z 695.480,A 0.000,B 0.000,C 90.000,E1 266.445} C_DIS
LIN {X 0.060,Y -426.038,Z 695.480,A 0.000,B 0.000,C 90.000,E1 266.331} C_DIS
LIN {X 0.149,Y -421.237,Z 695.479,A 0.000,B 0.000,C 90.000,E1 266.274} C_DIS
LIN {X -0.050,Y -414.821,Z 695.479,A 0.000,B 0.000,C 90.000,E1 266.274} C_DIS
LIN {X -0.044,Y -180.932,Z 695.479,A 0.000,B 0.000,C 90.000,E1 266.274} C_DIS
LIN {X -0.008,Y -180.776,Z 695.471,A 0.000,B 0.000,C 90.000,E1 264.723} C_DIS
LIN {X 0.030,Y -178.991,Z 695.444,A 0.000,B 0.000,C 90.000,E1 259.982} C_DIS
LIN {X 0.041,Y -177.976,Z 695.435,A 0.000,B 0.000,C 90.000,E1 258.285} C_DIS
LIN {X 0.011,Y -175.620,Z 695.411,A 0.000,B 0.000,C 90.000,E1 254.047} C_DIS
LIN {X 0.071,Y -172.341,Z 695.388,A 0.000,B 0.000,C 90.000,E1 249.752} C_DIS
LIN {X 0.050,Y -171.817,Z 695.383,A 0.000,B 0.000,C 90.000,E1 248.901} C_DIS
LIN {X 0.057,Y -170.284,Z 695.373,A 0.000,B 0.000,C 90.000,E1 247.177} C_DIS
LIN {X -0.008,Y -166.824,Z 695.349,A 0.000,B 0.000,C 90.000,E1 242.871} C_DIS
LIN {X -0.090,Y -162.806,Z 695.325,A 0.000,B 0.000,C 90.000,E1 238.535} C_DIS
LIN {X -0.025,Y -161.492,Z 695.315,A 0.000,B 0.000,C 90.000,E1 236.755} C_DIS
LIN {X 0.025,Y -157.489,Z 695.291,A 0.000,B 0.000,C 90.000,E1 232.316} C_DIS
LIN {X -0.037,Y -155.507,Z 695.276,A 0.000,B 0.000,C 90.000,E1 229.666} C_DIS
LIN {X 0.013,Y -151.809,Z 695.251,A 0.000,B 0.000,C 90.000,E1 225.162} C_DIS
LIN {X 0.026,Y -150.021,Z 695.236,A 0.000,B 0.000,C 90.000,E1 222.447} C_DIS
LIN {X 0.056,Y -146.843,Z 695.211,A 0.000,B 0.000,C 90.000,E1 217.890} C_DIS
LIN {X -0.041,Y -145.425,Z 695.195,A 0.000,B 0.000,C 90.000,E1 215.185} C_DIS
LIN {X -0.046,Y -142.851,Z 695.170,A 0.000,B 0.000,C 90.000,E1 210.590} C_DIS
LIN {X 0.007,Y -141.466,Z 695.149,A 0.000,B 0.000,C 90.000,E1 206.873} C_DIS
LIN {X -0.002,Y -139.377,Z 695.113,A 0.000,B 0.000,C 90.000,E1 200.375} C_DIS
LIN {X -0.012,Y -138.828,Z 695.098,A 0.000,B 0.000,C 90.000,E1 197.583} C_DIS
LIN {X 0.053,Y -138.353,Z 695.056,A 0.000,B 0.000,C 90.000,E1 190.084} C_DIS
LIN {X 0.050,Y -139.528,Z 695.004,A 0.000,B 0.000,C 90.000,E1 180.745} C_DIS
LIN {X 0.004,Y -141.204,Z 694.973,A 0.000,B 0.000,C 90.000,E1 175.179} C_DIS
LIN {X -0.037,Y -142.579,Z 694.958,A 0.000,B 0.000,C 90.000,E1 172.413} C_DIS
LIN {X 0.059,Y -144.873,Z 694.932,A 0.000,B 0.000,C 90.000,E1 167.757} C_DIS
LIN {X 0.013,Y -147.499,Z 694.912,A 0.000,B 0.000,C 90.000,E1 164.102} C_DIS
LIN {X 0.088,Y -150.091,Z 694.891,A 0.000,B 0.000,C 90.000,E1 160.423} C_DIS
LIN {X -0.041,Y -153.444,Z 694.871,A 0.000,B 0.000,C 90.000,E1 156.847} C_DIS
LIN {X -0.047,Y -157.807,Z 694.846,A 0.000,B 0.000,C 90.000,E1 152.359} C_DIS
LIN {X -0.015,Y -162.088,Z 694.827,A 0.000,B 0.000,C 90.000,E1 148.791} C_DIS
LIN {X 0.010,Y -166.288,Z 694.807,A 0.000,B 0.000,C 90.000,E1 145.261} C_DIS
LIN {X 0.007,Y -171.306,Z 694.788,A 0.000,B 0.000,C 90.000,E1 141.778} C_DIS
LIN {X 0.043,Y -176.202,Z 694.769,A 0.000,B 0.000,C 90.000,E1 138.324} C_DIS
LIN {X -0.092,Y -180.478,Z 694.754,A 0.000,B 0.000,C 90.000,E1 135.810} C_DIS
LIN {X 0.018,Y -185.882,Z 694.736,A 0.000,B 0.000,C 90.000,E1 132.405} C_DIS
LIN {X 0.052,Y -191.292,Z 694.719,A 0.000,B 0.000,C 90.000,E1 129.439} C_DIS
LIN {X 0.045,Y -289.146,Z 694.719,A 0.000,B 0.000,C 90.000,E1 129.439} C_DIS
LIN {X -0.063,Y -294.731,Z 694.718,A 0.000,B 0.000,C 90.000,E1 129.277} C_DIS
LIN {X 0.057,Y -297.167,Z 694.717,A 0.000,B 0.000,C 90.000,E1 129.072} C_DIS
LIN {X 0.061,Y -301.002,Z 694.715,A 0.000,B 0.000,C 90.000,E1 128.624} C_DIS
LIN {X 0.080,Y -302.894,Z 694.713,A 0.000,B 0.000,C 90.000,E1 128.302} C_DIS
LIN {X -0.092,Y -304.378,Z 694.711,A 0.000,B 0.000,C 90.000,E1 128.016} C_DIS
LIN {X 0.109,Y -305.590,Z 694.709,A 0.000,B 0.000,C 90.000,E1 127.649} C_DIS
LIN {X -0.141,Y -317.273,Z 694.688,A 0.000,B 0.000,C 90.000,E1 123.785} C_DIS
LIN {X 0.059,Y -327.416,Z 694.672,A 0.000,B 0.000,C 90.000,E1 120.875} C_DIS
LIN {X 0.067,Y -338.891,Z 694.656,A 0.000,B 0.000,C 90.000,E1 118.052} C_DIS
LIN {X 0.083,Y -351.807,Z 694.641,A 0.000,B 0.000,C 90.000,E1 115.283} C_DIS
LIN {X -0.056,Y -364.585,Z 694.627,A 0.000,B 0.000,C 90.000,E1 112.898} C_DIS
LIN {X -0.163,Y -378.681,Z 694.614,A 0.000,B 0.000,C 90.000,E1 110.556} C_DIS
LIN {X -0.057,Y -394.197,Z 694.601,A 0.000,B 0.000,C 90.000,E1 108.236} C_DIS
LIN {X 0.075,Y -411.245,Z 694.589,A 0.000,B 0.000,C 90.000,E1 105.969} C_DIS
LIN {X 0.135,Y -429.951,Z 694.577,A 0.000,B 0.000,C 90.000,E1 103.772} C_DIS
LIN {X -0.024,Y -449.942,Z 694.565,A 0.000,B 0.000,C 90.000,E1 101.715} C_DIS
LIN {X 0.149,Y -467.883,Z 694.556,A 0.000,B 0.000,C 90.000,E1 100.018} C_DIS
LIN {X 0.111,Y -470.189,Z 694.555,A 0.000,B 0.000,C 90.000,E1 99.792} C_DIS
LIN {X 0.012,Y -472.037,Z 694.553,A 0.000,B 0.000,C 90.000,E1 99.557} C_DIS
LIN {X -0.087,Y -473.433,Z 694.552,A 0.000,B 0.000,C 90.000,E1 99.321} C_DIS
LIN {X 0.023,Y -475.258,Z 694.549,A 0.000,B 0.000,C 90.000,E1 98.803} C_DIS
LIN {X 0.214,Y -475.987,Z 694.546,A 0.000,B 0.000,C 90.000,E1 98.276} C_DIS
LIN {X -0.127,Y -475.747,Z 694.543,A 0.000,B 0.000,C 90.000,E1 97.814} C_DIS
LIN {X 0.010,Y -474.505,Z 694.541,A 0.000,B 0.000,C 90.000,E1 97.296} C_DIS
LIN {X -0.187,Y -473.448,Z 694.539,A 0.000,B 0.000,C 90.000,E1 97.068} C_DIS
LIN {X 0.144,Y -472.032,Z 694.538,A 0.000,B 0.000,C 90.000,E1 96.777} C_DIS
LIN {X 0.076,Y -452.270,Z 694.521,A 0.000,B 0.000,C 90.000,E1 93.726} C_DIS
LIN {X -0.165,Y -437.585,Z 694.506,A 0.000,B 0.000,C 90.000,E1 91.146} C_DIS
LIN {X -0.083,Y -428.672,Z 694.497,A 0.000,B 0.000,C 90.000,E1 89.542} C_DIS
LIN {X -0.149,Y -419.418,Z 694.488,A 0.000,B 0.000,C 90.000,E1 87.936} C_DIS
LIN {X 0.112,Y -408.439,Z 694.478,A 0.000,B 0.000,C 90.000,E1 85.988} C_DIS
LIN {X -0.136,Y -395.930,Z 694.465,A 0.000,B 0.000,C 90.000,E1 83.799} C_DIS
LIN {X -0.213,Y -380.672,Z 694.450,A 0.000,B 0.000,C 90.000,E1 80.971} C_DIS
LIN {X -0.106,Y -368.968,Z 694.437,A 0.000,B 0.000,C 90.000,E1 78.634} C_DIS
LIN {X 0.014,Y -353.440,Z 694.419,A 0.000,B 0.000,C 90.000,E1 75.353} C_DIS
LIN {X 0.053,Y -340.059,Z 694.402,A 0.000,B 0.000,C 90.000,E1 72.308} C_DIS
LIN {X -0.027,Y -325.991,Z 694.383,A 0.000,B 0.000,C 90.000,E1 68.901} C_DIS
LIN {X -0.066,Y -315.501,Z 694.367,A 0.000,B 0.000,C 90.000,E1 66.049} C_DIS
LIN {X -0.007,Y -303.316,Z 694.345,A 0.000,B 0.000,C 90.000,E1 62.153} C_DIS
LIN {X -0.089,Y -294.071,Z 694.327,A 0.000,B 0.000,C 90.000,E1 58.869} C_DIS
LIN {X -0.092,Y -285.417,Z 694.308,A 0.000,B 0.000,C 90.000,E1 55.515} C_DIS
LIN {X 0.051,Y -278.743,Z 694.293,A 0.000,B 0.000,C 90.000,E1 52.763} C_DIS
LIN {X -0.064,Y -273.566,Z 694.282,A 0.000,B 0.000,C 90.000,E1 50.723} C_DIS
LIN {X 0.073,Y -268.226,Z 694.270,A 0.000,B 0.000,C 90.000,E1 48.609} C_DIS
LIN {X -0.094,Y -262.518,Z 694.258,A 0.000,B 0.000,C 90.000,E1 46.539} C_DIS
LIN {X -0.015,Y -256.572,Z 694.247,A 0.000,B 0.000,C 90.000,E1 44.393} C_DIS
LIN {X -0.033,Y -250.513,Z 694.235,A 0.000,B 0.000,C 90.000,E1 42.243} C_DIS
LIN {X -0.155,Y -244.273,Z 694.223,A 0.000,B 0.000,C 90.000,E1 40.092} C_DIS
LIN {X -0.066,Y -234.110,Z 694.202,A 0.000,B 0.000,C 90.000,E1 36.377} C_DIS
LIN {X -0.085,Y -226.511,Z 694.185,A 0.000,B 0.000,C 90.000,E1 33.372} C_DIS
LIN {X 0.031,Y -219.625,Z 694.168,A 0.000,B 0.000,C 90.000,E1 30.285} C_DIS
LIN {X -0.051,Y -213.573,Z 694.151,A 0.000,B 0.000,C 90.000,E1 27.206} C_DIS
LIN {X -0.099,Y -208.314,Z 694.134,A 0.000,B 0.000,C 90.000,E1 24.079} C_DIS
LIN {X 0.037,Y -202.909,Z 694.112,A 0.000,B 0.000,C 90.000,E1 20.066} C_DIS
LIN {X -0.076,Y -198.668,Z 694.089,A 0.000,B 0.000,C 90.000,E1 16.079} C_DIS
LIN {X 0.003,Y -195.025,Z 694.062,A 0.000,B 0.000,C 90.000,E1 11.186} C_DIS
LIN {X -0.011,Y -192.490,Z 694.026,A 0.000,B 0.000,C 90.000,E1 4.645} C_DIS
LIN {X -0.044,Y -193.986,Z 693.965,A 0.000,B 0.000,C 90.000,E1 353.799} C_DIS
LIN {X 0.046,Y -196.975,Z 693.938,A 0.000,B 0.000,C 90.000,E1 348.870} C_DIS
LIN {X 0.051,Y -200.550,Z 693.916,A 0.000,B 0.000,C 90.000,E1 344.810} C_DIS
LIN {X 0.052,Y -205.100,Z 693.893,A 0.000,B 0.000,C 90.000,E1 340.786} C_DIS
LIN {X 0.083,Y -210.500,Z 693.871,A 0.000,B 0.000,C 90.000,E1 336.794} C_DIS
LIN {X 0.034,Y -216.597,Z 693.849,A 0.000,B 0.000,C 90.000,E1 332.871} C_DIS
LIN {X -0.002,Y -223.435,Z 693.828,A 0.000,B 0.000,C 90.000,E1 328.997} C_DIS
LIN {X -0.052,Y -230.910,Z 693.807,A 0.000,B 0.000,C 90.000,E1 325.182} C_DIS
LIN {X -0.045,Y -238.993,Z 693.786,A 0.000,B 0.000,C 90.000,E1 321.412} C_DIS
LIN {X -0.082,Y -247.974,Z 693.765,A 0.000,B 0.000,C 90.000,E1 317.715} C_DIS
LIN {X -0.051,Y -256.938,Z 693.747,A 0.000,B 0.000,C 90.000,E1 314.433} C_DIS
LIN {X -0.028,Y -267.970,Z 693.727,A 0.000,B 0.000,C 90.000,E1 310.862} C_DIS
LIN {X -0.076,Y -279.060,Z 693.710,A 0.000,B 0.000,C 90.000,E1 307.729} C_DIS
LIN {X -0.128,Y -292.667,Z 693.691,A 0.000,B 0.000,C 90.000,E1 304.326} C_DIS
LIN {X -0.155,Y -307.752,Z 693.672,A 0.000,B 0.000,C 90.000,E1 301.003} C_DIS
LIN {X 0.110,Y -320.867,Z 693.658,A 0.000,B 0.000,C 90.000,E1 298.359} C_DIS
LIN {X -0.027,Y -334.941,Z 693.644,A 0.000,B 0.000,C 90.000,E1 295.848} C_DIS
LIN {X -0.110,Y -349.827,Z 693.630,A 0.000,B 0.000,C 90.000,E1 293.387} C_DIS
LIN {X -0.030,Y -367.489,Z 693.615,A 0.000,B 0.000,C 90.000,E1 290.663} C_DIS
LIN {X -0.188,Y -377.965,Z 693.607,A 0.000,B 0.000,C 90.000,E1 289.214} C_DIS
LIN {X -0.163,Y -398.602,Z 693.592,A 0.000,B 0.000,C 90.000,E1 286.622} C_DIS
LIN {X 0.155,Y -412.511,Z 693.583,A 0.000,B 0.000,C 90.000,E1 284.898} C_DIS
LIN {X 0.079,Y -423.892,Z 693.575,A 0.000,B 0.000,C 90.000,E1 283.536} C_DIS
LIN {X 0.077,Y -434.819,Z 693.568,A 0.000,B 0.000,C 90.000,E1 282.187} C_DIS
LIN {X -0.203,Y -445.131,Z 693.560,A 0.000,B 0.000,C 90.000,E1 280.894} C_DIS
LIN {X -0.209,Y -463.043,Z 693.547,A 0.000,B 0.000,C 90.000,E1 278.568} C_DIS
LIN {X -0.090,Y -470.918,Z 693.542,A 0.000,B 0.000,C 90.000,E1 277.530} C_DIS
LIN {X -0.145,Y -476.207,Z 693.538,A 0.000,B 0.000,C 90.000,E1 276.777} C_DIS
LIN {X -0.015,Y -479.245,Z 693.535,A 0.000,B 0.000,C 90.000,E1 276.258} C_DIS
LIN {X 0.136,Y -481.854,Z 693.532,A 0.000,B 0.000,C 90.000,E1 275.739} C_DIS
LIN {X -0.179,Y -484.002,Z 693.529,A 0.000,B 0.000,C 90.000,E1 275.277} C_DIS
LIN {X -0.001,Y -485.721,Z 693.526,A 0.000,B 0.000,C 90.000,E1 274.759} C_DIS
LIN {X 0.146,Y -486.982,Z 693.524,A 0.000,B 0.000,C 90.000,E1 274.245} C_DIS
LIN {X -0.145,Y -487.877,Z 693.521,A 0.000,B 0.000,C 90.000,E1 273.784} C_DIS
LIN {X 0.025,Y -488.366,Z 693.518,A 0.000,B 0.000,C 90.000,E1 273.269} C_DIS
LIN {X 0.228,Y -488.516,Z 693.515,A 0.000,B 0.000,C 90.000,E1 272.751} C_DIS
LIN {X -0.078,Y -488.353,Z 693.513,A 0.000,B 0.000,C 90.000,E1 272.293} C_DIS
LIN {X 0.123,Y -487.853,Z 693.510,A 0.000,B 0.000,C 90.000,E1 271.776} C_DIS
LIN {X -0.182,Y -486.994,Z 693.507,A 0.000,B 0.000,C 90.000,E1 271.318} C_DIS
LIN {X 0.000,Y -485.762,Z 693.504,A 0.000,B 0.000,C 90.000,E1 270.802} C_DIS
LIN {X 0.176,Y -484.011,Z 693.502,A 0.000,B 0.000,C 90.000,E1 270.286} C_DIS
LIN {X -0.138,Y -481.680,Z 693.499,A 0.000,B 0.000,C 90.000,E1 269.828} C_DIS
LIN {X 0.180,Y -480.347,Z 693.498,A 0.000,B 0.000,C 90.000,E1 269.542} C_DIS
LIN {X -0.156,Y -477.014,Z 693.495,A 0.000,B 0.000,C 90.000,E1 269.083} C_DIS
LIN {X -0.030,Y -472.792,Z 693.492,A 0.000,B 0.000,C 90.000,E1 268.568} C_DIS
LIN {X 0.116,Y -467.591,Z 693.489,A 0.000,B 0.000,C 90.000,E1 268.051} C_DIS
LIN {X -0.043,Y -464.528,Z 693.488,A 0.000,B 0.000,C 90.000,E1 267.822} C_DIS
LIN {X 0.153,Y -457.996,Z 693.485,A 0.000,B 0.000,C 90.000,E1 267.364} C_DIS
LIN {X 0.085,Y -454.711,Z 693.484,A 0.000,B 0.000,C 90.000,E1 267.192} C_DIS
LIN {X -0.186,Y -447.569,Z 693.483,A 0.000,B 0.000,C 90.000,E1 266.906} C_DIS
LIN {X 0.069,Y -440.365,Z 693.481,A 0.000,B 0.000,C 90.000,E1 266.617} C_DIS
LIN {X 0.057,Y -436.216,Z 693.481,A 0.000,B 0.000,C 90.000,E1 266.502} C_DIS
LIN {X -0.172,Y -431.980,Z 693.480,A 0.000,B 0.000,C 90.000,E1 266.445} C_DIS
LIN {X 0.119,Y -421.611,Z 693.479,A 0.000,B 0.000,C 90.000,E1 266.274} C_DIS
LIN {X -0.080,Y -416.282,Z 693.479,A 0.000,B 0.000,C 90.000,E1 266.274} C_DIS
LIN {X -0.057,Y -180.932,Z 693.479,A 0.000,B 0.000,C 90.000,E1 266.274} C_DIS
LIN {X -0.021,Y -180.774,Z 693.471,A 0.000,B 0.000,C 90.000,E1 264.723} C_DIS
LIN {X 0.017,Y -178.989,Z 693.444,A 0.000,B 0.000,C 90.000,E1 259.982} C_DIS
LIN {X 0.027,Y -177.973,Z 693.435,A 0.000,B 0.000,C 90.000,E1 258.285} C_DIS
LIN {X 0.046,Y -175.616,Z 693.411,A 0.000,B 0.000,C 90.000,E1 254.031} C_DIS
LIN {X 0.058,Y -172.338,Z 693.388,A 0.000,B 0.000,C 90.000,E1 249.752} C_DIS
LIN {X 0.037,Y -171.814,Z 693.383,A 0.000,B 0.000,C 90.000,E1 248.901} C_DIS
LIN {X 0.043,Y -170.280,Z 693.373,A 0.000,B 0.000,C 90.000,E1 247.177} C_DIS
LIN {X -0.021,Y -166.820,Z 693.349,A 0.000,B 0.000,C 90.000,E1 242.871} C_DIS
LIN {X 0.036,Y -162.802,Z 693.325,A 0.000,B 0.000,C 90.000,E1 238.486} C_DIS
LIN {X -0.038,Y -161.489,Z 693.315,A 0.000,B 0.000,C 90.000,E1 236.755} C_DIS
LIN {X 0.012,Y -157.485,Z 693.291,A 0.000,B 0.000,C 90.000,E1 232.316} C_DIS
LIN {X -0.050,Y -155.503,Z 693.276,A 0.000,B 0.000,C 90.000,E1 229.666} C_DIS
LIN {X 0.001,Y -151.806,Z 693.251,A 0.000,B 0.000,C 90.000,E1 225.162} C_DIS
LIN {X 0.013,Y -150.017,Z 693.236,A 0.000,B 0.000,C 90.000,E1 222.447} C_DIS
LIN {X 0.044,Y -146.841,Z 693.211,A 0.000,B 0.000,C 90.000,E1 217.890} C_DIS
LIN {X 0.031,Y -145.423,Z 693.195,A 0.000,B 0.000,C 90.000,E1 215.152} C_DIS
LIN {X -0.057,Y -142.849,Z 693.170,A 0.000,B 0.000,C 90.000,E1 210.590} C_DIS
LIN {X -0.004,Y -141.463,Z 693.149,A 0.000,B 0.000,C 90.000,E1 206.873} C_DIS
LIN {X -0.013,Y -139.376,Z 693.113,A 0.000,B 0.000,C 90.000,E1 200.375} C_DIS
LIN {X -0.023,Y -138.827,Z 693.098,A 0.000,B 0.000,C 90.000,E1 197.583} C_DIS
LIN {X 0.041,Y -138.353,Z 693.056,A 0.000,B 0.000,C 90.000,E1 190.084} C_DIS
LIN {X 0.039,Y -139.529,Z 693.004,A 0.000,B 0.000,C 90.000,E1 180.745} C_DIS
LIN {X -0.008,Y -141.206,Z 692.973,A 0.000,B 0.000,C 90.000,E1 175.179} C_DIS
LIN {X -0.049,Y -142.582,Z 692.958,A 0.000,B 0.000,C 90.000,E1 172.413} C_DIS
LIN {X 0.047,Y -144.876,Z 692.932,A 0.000,B 0.000,C 90.000,E1 167.757} C_DIS
LIN {X 0.000,Y -147.503,Z 692.912,A 0.000,B 0.000,C 90.000,E1 164.102} C_DIS
LIN {X 0.075,Y -150.094,Z 692.891,A 0.000,B 0.000,C 90.000,E1 160.423} C_DIS
LIN {X 0.088,Y -153.449,Z 692.871,A 0.000,B 0.000,C 90.000,E1 156.794} C_DIS
LIN {X -0.060,Y -157.812,Z 692.846,A 0.000,B 0.000,C 90.000,E1 152.359} C_DIS
LIN {X -0.028,Y -162.094,Z 692.827,A 0.000,B 0.000,C 90.000,E1 148.791} C_DIS
LIN {X -0.003,Y -166.294,Z 692.807,A 0.000,B 0.000,C 90.000,E1 145.261} C_DIS
LIN {X -0.006,Y -171.312,Z 692.788,A 0.000,B 0.000,C 90.000,E1 141.778} C_DIS
LIN {X 0.029,Y -176.209,Z 692.768,A 0.000,B 0.000,C 90.000,E1 138.324} C_DIS
LIN {X -0.107,Y -180.486,Z 692.754,A 0.000,B 0.000,C 90.000,E1 135.810} C_DIS
LIN {X 0.005,Y -185.890,Z 692.736,A 0.000,B 0.000,C 90.000,E1 132.405} C_DIS
LIN {X -0.063,Y -191.276,Z 692.719,A 0.000,B 0.000,C 90.000,E1 129.483} C_DIS
LIN {X -0.130,Y -289.507,Z 692.719,A 0.000,B 0.000,C 90.000,E1 129.483} C_DIS
LIN {X 0.024,Y -290.485,Z 692.719,A 0.000,B 0.000,C 90.000,E1 129.439} C_DIS
LIN {X -0.085,Y -294.943,Z 692.718,A 0.000,B 0.000,C 90.000,E1 129.277} C_DIS
LIN {X 0.035,Y -297.296,Z 692.717,A 0.000,B 0.000,C 90.000,E1 129.072} C_DIS
LIN {X -0.033,Y -301.148,Z 692.715,A 0.000,B 0.000,C 90.000,E1 128.624} C_DIS
LIN {X -0.046,Y -303.025,Z 692.713,A 0.000,B 0.000,C 90.000,E1 128.302} C_DIS
LIN {X -0.009,Y -304.495,Z 692.711,A 0.000,B 0.000,C 90.000,E1 127.971} C_DIS
LIN {X -0.049,Y -305.670,Z 692.709,A 0.000,B 0.000,C 90.000,E1 127.649} C_DIS
LIN {X 0.074,Y -316.299,Z 692.689,A 0.000,B 0.000,C 90.000,E1 124.040} C_DIS
LIN {X -0.033,Y -326.310,Z 692.673,A 0.000,B 0.000,C 90.000,E1 121.180} C_DIS
LIN {X -0.077,Y -337.648,Z 692.657,A 0.000,B 0.000,C 90.000,E1 118.359} C_DIS
LIN {X -0.106,Y -350.409,Z 692.642,A 0.000,B 0.000,C 90.000,E1 115.591} C_DIS
LIN {X 0.043,Y -363.043,Z 692.629,A 0.000,B 0.000,C 90.000,E1 113.153} C_DIS
LIN {X 0.040,Y -376.984,Z 692.616,A 0.000,B 0.000,C 90.000,E1 110.791} C_DIS
LIN {X -0.020,Y -392.333,Z 692.603,A 0.000,B 0.000,C 90.000,E1 108.489} C_DIS
LIN {X -0.201,Y -409.201,Z 692.590,A 0.000,B 0.000,C 90.000,E1 106.260} C_DIS
LIN {X -0.210,Y -427.711,Z 692.578,A 0.000,B 0.000,C 90.000,E1 104.064} C_DIS
LIN {X -0.086,Y -447.602,Z 692.566,A 0.000,B 0.000,C 90.000,E1 101.951} C_DIS
LIN {X -0.027,Y -468.095,Z 692.556,A 0.000,B 0.000,C 90.000,E1 100.018} C_DIS
LIN {X -0.064,Y -470.361,Z 692.554,A 0.000,B 0.000,C 90.000,E1 99.792} C_DIS
LIN {X -0.183,Y -472.196,Z 692.553,A 0.000,B 0.000,C 90.000,E1 99.557} C_DIS
LIN {X 0.164,Y -473.579,Z 692.552,A 0.000,B 0.000,C 90.000,E1 99.265} C_DIS
LIN {X -0.193,Y -475.361,Z 692.549,A 0.000,B 0.000,C 90.000,E1 98.803} C_DIS
LIN {X -0.001,Y -476.056,Z 692.546,A 0.000,B 0.000,C 90.000,E1 98.276} C_DIS
LIN {X 0.130,Y -475.784,Z 692.543,A 0.000,B 0.000,C 90.000,E1 97.757} C_DIS
LIN {X -0.204,Y -474.504,Z 692.540,A 0.000,B 0.000,C 90.000,E1 97.296} C_DIS
LIN {X 0.128,Y -473.425,Z 692.539,A 0.000,B 0.000,C 90.000,E1 97.004} C_DIS
LIN {X -0.068,Y -471.980,Z 692.538,A 0.000,B 0.000,C 90.000,E1 96.777} C_DIS
LIN {X 0.102,Y -453.749,Z 692.522,A 0.000,B 0.000,C 90.000,E1 93.955} C_DIS
LIN {X 0.072,Y -437.524,Z 692.506,A 0.000,B 0.000,C 90.000,E1 91.088} C_DIS
LIN {X 0.147,Y -428.621,Z 692.497,A 0.000,B 0.000,C 90.000,E1 89.484} C_DIS
LIN {X 0.076,Y -419.353,Z 692.488,A 0.000,B 0.000,C 90.000,E1 87.879} C_DIS
LIN {X -0.079,Y -408.386,Z 692.478,A 0.000,B 0.000,C 90.000,E1 85.988} C_DIS
LIN {X 0.071,Y -395.879,Z 692.465,A 0.000,B 0.000,C 90.000,E1 83.742} C_DIS
LIN {X 0.042,Y -380.650,Z 692.450,A 0.000,B 0.000,C 90.000,E1 80.905} C_DIS
LIN {X 0.081,Y -368.954,Z 692.437,A 0.000,B 0.000,C 90.000,E1 78.578} C_DIS
LIN {X -0.065,Y -353.460,Z 692.418,A 0.000,B 0.000,C 90.000,E1 75.338} C_DIS
LIN {X -0.107,Y -340.096,Z 692.402,A 0.000,B 0.000,C 90.000,E1 72.308} C_DIS
LIN {X -0.180,Y -326.093,Z 692.383,A 0.000,B 0.000,C 90.000,E1 68.901} C_DIS
LIN {X 0.078,Y -315.638,Z 692.367,A 0.000,B 0.000,C 90.000,E1 65.997} C_DIS
LIN {X 0.128,Y -303.479,Z 692.345,A 0.000,B 0.000,C 90.000,E1 62.103} C_DIS
LIN {X 0.038,Y -294.253,Z 692.327,A 0.000,B 0.000,C 90.000,E1 58.820} C_DIS
LIN {X 0.028,Y -285.634,Z 692.308,A 0.000,B 0.000,C 90.000,E1 55.468} C_DIS
LIN {X -0.056,Y -278.964,Z 692.293,A 0.000,B 0.000,C 90.000,E1 52.763} C_DIS
LIN {X 0.047,Y -273.825,Z 692.282,A 0.000,B 0.000,C 90.000,E1 50.678} C_DIS
LIN {X -0.022,Y -268.454,Z 692.270,A 0.000,B 0.000,C 90.000,E1 48.609} C_DIS
LIN {X -0.003,Y -262.736,Z 692.258,A 0.000,B 0.000,C 90.000,E1 46.500} C_DIS
LIN {X 0.087,Y -256.760,Z 692.247,A 0.000,B 0.000,C 90.000,E1 44.352} C_DIS
LIN {X 0.058,Y -250.689,Z 692.235,A 0.000,B 0.000,C 90.000,E1 42.204} C_DIS
LIN {X 0.117,Y -244.455,Z 692.222,A 0.000,B 0.000,C 90.000,E1 40.011} C_DIS
LIN {X 0.058,Y -236.229,Z 692.206,A 0.000,B 0.000,C 90.000,E1 37.076} C_DIS
LIN {X -0.143,Y -226.631,Z 692.185,A 0.000,B 0.000,C 90.000,E1 33.372} C_DIS
LIN {X 0.088,Y -219.762,Z 692.168,A 0.000,B 0.000,C 90.000,E1 30.256} C_DIS
LIN {X -0.002,Y -213.688,Z 692.151,A 0.000,B 0.000,C 90.000,E1 27.180} C_DIS
LIN {X 0.046,Y -208.454,Z 692.134,A 0.000,B 0.000,C 90.000,E1 24.027} C_DIS
LIN {X -0.002,Y -203.045,Z 692.111,A 0.000,B 0.000,C 90.000,E1 20.066} C_DIS
LIN {X 0.081,Y -198.828,Z 692.089,A 0.000,B 0.000,C 90.000,E1 16.024} C_DIS
LIN {X -0.024,Y -195.183,Z 692.062,A 0.000,B 0.000,C 90.000,E1 11.186} C_DIS
LIN {X -0.031,Y -192.640,Z 692.026,A 0.000,B 0.000,C 90.000,E1 4.645} C_DIS
LIN {X -0.038,Y -194.096,Z 691.966,A 0.000,B 0.000,C 90.000,E1 353.799} C_DIS
LIN {X 0.080,Y -197.696,Z 691.934,A 0.000,B 0.000,C 90.000,E1 348.049} C_DIS
LIN {X -0.036,Y -201.458,Z 691.911,A 0.000,B 0.000,C 90.000,E1 344.031} C_DIS
LIN {X -0.010,Y -206.166,Z 691.889,A 0.000,B 0.000,C 90.000,E1 340.007} C_DIS
LIN {X -0.070,Y -211.724,Z 691.867,A 0.000,B 0.000,C 90.000,E1 336.049} C_DIS
LIN {X 0.007,Y -217.946,Z 691.845,A 0.000,B 0.000,C 90.000,E1 332.103} C_DIS
LIN {X -0.071,Y -224.943,Z 691.823,A 0.000,B 0.000,C 90.000,E1 328.250} C_DIS
LIN {X 0.057,Y -232.523,Z 691.802,A 0.000,B 0.000,C 90.000,E1 324.402} C_DIS
LIN {X 0.080,Y -240.742,Z 691.781,A 0.000,B 0.000,C 90.000,E1 320.642} C_DIS
LIN {X -0.073,Y -249.903,Z 691.761,A 0.000,B 0.000,C 90.000,E1 316.986} C_DIS
LIN {X 0.025,Y -259.065,Z 691.743,A 0.000,B 0.000,C 90.000,E1 313.704} C_DIS
LIN {X -0.135,Y -269.140,Z 691.725,A 0.000,B 0.000,C 90.000,E1 310.539} C_DIS
LIN {X 0.065,Y -280.351,Z 691.708,A 0.000,B 0.000,C 90.000,E1 307.363} C_DIS
LIN {X -0.108,Y -294.112,Z 691.689,A 0.000,B 0.000,C 90.000,E1 303.992} C_DIS
LIN {X -0.082,Y -309.326,Z 691.670,A 0.000,B 0.000,C 90.000,E1 300.669} C_DIS
LIN {X 0.147,Y -320.873,Z 691.658,A 0.000,B 0.000,C 90.000,E1 298.359} C_DIS
LIN {X -0.014,Y -336.722,Z 691.642,A 0.000,B 0.000,C 90.000,E1 295.540} C_DIS
LIN {X -0.024,Y -353.569,Z 691.626,A 0.000,B 0.000,C 90.000,E1 292.770} C_DIS
LIN {X 0.129,Y -373.534,Z 691.610,A 0.000,B 0.000,C 90.000,E1 289.758} C_DIS
LIN {X 0.082,Y -384.514,Z 691.602,A 0.000,B 0.000,C 90.000,E1 288.308} C_DIS
LIN {X 0.041,Y -400.755,Z 691.591,A 0.000,B 0.000,C 90.000,E1 286.315} C_DIS
LIN {X -0.211,Y -412.350,Z 691.583,A 0.000,B 0.000,C 90.000,E1 284.954} C_DIS
LIN {X 0.110,Y -423.723,Z 691.575,A 0.000,B 0.000,C 90.000,E1 283.536} C_DIS
LIN {X 0.107,Y -434.665,Z 691.568,A 0.000,B 0.000,C 90.000,E1 282.187} C_DIS
LIN {X -0.175,Y -444.945,Z 691.560,A 0.000,B 0.000,C 90.000,E1 280.894} C_DIS
LIN {X 0.140,Y -462.946,Z 691.547,A 0.000,B 0.000,C 90.000,E1 278.511} C_DIS
LIN {X -0.202,Y -470.842,Z 691.542,A 0.000,B 0.000,C 90.000,E1 277.530} C_DIS
LIN {X 0.214,Y -476.122,Z 691.537,A 0.000,B 0.000,C 90.000,E1 276.720} C_DIS
LIN {X -0.130,Y -479.139,Z 691.535,A 0.000,B 0.000,C 90.000,E1 276.258} C_DIS
LIN {X 0.019,Y -481.747,Z 691.532,A 0.000,B 0.000,C 90.000,E1 275.739} C_DIS
LIN {X 0.185,Y -483.876,Z 691.529,A 0.000,B 0.000,C 90.000,E1 275.220} C_DIS
LIN {X -0.120,Y -485.564,Z 691.526,A 0.000,B 0.000,C 90.000,E1 274.759} C_DIS
LIN {X 0.026,Y -486.823,Z 691.524,A 0.000,B 0.000,C 90.000,E1 274.245} C_DIS
LIN {X 0.220,Y -487.727,Z 691.521,A 0.000,B 0.000,C 90.000,E1 273.726} C_DIS
LIN {X -0.098,Y -488.207,Z 691.518,A 0.000,B 0.000,C 90.000,E1 273.269} C_DIS
LIN {X 0.105,Y -488.354,Z 691.515,A 0.000,B 0.000,C 90.000,E1 272.751} C_DIS
LIN {X -0.202,Y -488.208,Z 691.513,A 0.000,B 0.000,C 90.000,E1 272.293} C_DIS
LIN {X -0.002,Y -487.721,Z 691.510,A 0.000,B 0.000,C 90.000,E1 271.776} C_DIS
LIN {X 0.179,Y -486.888,Z 691.507,A 0.000,B 0.000,C 90.000,E1 271.260} C_DIS
LIN {X -0.126,Y -485.632,Z 691.504,A 0.000,B 0.000,C 90.000,E1 270.802} C_DIS
LIN {X 0.050,Y -483.896,Z 691.502,A 0.000,B 0.000,C 90.000,E1 270.286} C_DIS
LIN {X 0.217,Y -481.604,Z 691.499,A 0.000,B 0.000,C 90.000,E1 269.771} C_DIS
LIN {X -0.112,Y -478.658,Z 691.496,A 0.000,B 0.000,C 90.000,E1 269.312} C_DIS
LIN {X 0.024,Y -474.925,Z 691.493,A 0.000,B 0.000,C 90.000,E1 268.797} C_DIS
LIN {X 0.137,Y -470.210,Z 691.491,A 0.000,B 0.000,C 90.000,E1 268.282} C_DIS
LIN {X -0.004,Y -467.468,Z 691.489,A 0.000,B 0.000,C 90.000,E1 268.051} C_DIS
LIN {X -0.157,Y -464.395,Z 691.488,A 0.000,B 0.000,C 90.000,E1 267.822} C_DIS
LIN {X 0.054,Y -457.794,Z 691.485,A 0.000,B 0.000,C 90.000,E1 267.364} C_DIS
LIN {X 0.010,Y -454.558,Z 691.484,A 0.000,B 0.000,C 90.000,E1 267.192} C_DIS
LIN {X 0.196,Y -447.435,Z 691.483,A 0.000,B 0.000,C 90.000,E1 266.849} C_DIS
LIN {X -0.002,Y -440.193,Z 691.481,A 0.000,B 0.000,C 90.000,E1 266.617} C_DIS
LIN {X -0.008,Y -435.949,Z 691.481,A 0.000,B 0.000,C 90.000,E1 266.502} C_DIS
LIN {X 0.212,Y -431.868,Z 691.480,A 0.000,B 0.000,C 90.000,E1 266.388} C_DIS
LIN {X 0.090,Y -421.740,Z 691.479,A 0.000,B 0.000,C 90.000,E1 266.274} C_DIS
LIN {X -0.155,Y -413.263,Z 691.479,A 0.000,B 0.000,C 90.000,E1 266.274} C_DIS
LIN {X -0.090,Y -180.932,Z 691.479,A 0.000,B 0.000,C 90.000,E1 266.274} C_DIS
LIN {X -0.032,Y -180.772,Z 691.471,A 0.000,B 0.000,C 90.000,E1 264.723} C_DIS
LIN {X 0.005,Y -178.988,Z 691.444,A 0.000,B 0.000,C 90.000,E1 259.982} C_DIS
LIN {X 0.016,Y -177.971,Z 691.435,A 0.000,B 0.000,C 90.000,E1 258.285} C_DIS
LIN {X 0.035,Y -175.614,Z 691.411,A 0.000,B 0.000,C 90.000,E1 254.031} C_DIS
LIN {X 0.047,Y -172.336,Z 691.388,A 0.000,B 0.000,C 90.000,E1 249.752} C_DIS
LIN {X 0.025,Y -171.812,Z 691.383,A 0.000,B 0.000,C 90.000,E1 248.901} C_DIS
LIN {X 0.033,Y -170.276,Z 691.373,A 0.000,B 0.000,C 90.000,E1 247.177} C_DIS
LIN {X -0.031,Y -166.817,Z 691.349,A 0.000,B 0.000,C 90.000,E1 242.871} C_DIS
LIN {X 0.026,Y -162.799,Z 691.325,A 0.000,B 0.000,C 90.000,E1 238.486} C_DIS
LIN {X -0.049,Y -161.487,Z 691.315,A 0.000,B 0.000,C 90.000,E1 236.755} C_DIS
LIN {X 0.002,Y -157.482,Z 691.291,A 0.000,B 0.000,C 90.000,E1 232.316} C_DIS
LIN {X 0.059,Y -155.499,Z 691.276,A 0.000,B 0.000,C 90.000,E1 229.622} C_DIS
LIN {X -0.009,Y -151.804,Z 691.251,A 0.000,B 0.000,C 90.000,E1 225.162} C_DIS
LIN {X 0.004,Y -150.014,Z 691.236,A 0.000,B 0.000,C 90.000,E1 222.447} C_DIS
LIN {X 0.034,Y -146.838,Z 691.211,A 0.000,B 0.000,C 90.000,E1 217.890} C_DIS
LIN {X 0.021,Y -145.420,Z 691.195,A 0.000,B 0.000,C 90.000,E1 215.152} C_DIS
LIN {X 0.056,Y -142.847,Z 691.170,A 0.000,B 0.000,C 90.000,E1 210.541} C_DIS
LIN {X -0.014,Y -141.461,Z 691.149,A 0.000,B 0.000,C 90.000,E1 206.873} C_DIS
LIN {X -0.023,Y -139.375,Z 691.113,A 0.000,B 0.000,C 90.000,E1 200.375} C_DIS
LIN {X -0.032,Y -138.826,Z 691.098,A 0.000,B 0.000,C 90.000,E1 197.583} C_DIS
LIN {X 0.055,Y -138.353,Z 691.056,A 0.000,B 0.000,C 90.000,E1 190.074} C_DIS
LIN {X 0.029,Y -139.530,Z 691.004,A 0.000,B 0.000,C 90.000,E1 180.745} C_DIS
LIN {X -0.018,Y -141.208,Z 690.973,A 0.000,B 0.000,C 90.000,E1 175.179} C_DIS
LIN {X -0.059,Y -142.583,Z 690.958,A 0.000,B 0.000,C 90.000,E1 172.413} C_DIS
LIN {X 0.036,Y -144.878,Z 690.932,A 0.000,B 0.000,C 90.000,E1 167.757} C_DIS
LIN {X -0.009,Y -147.506,Z 690.912,A 0.000,B 0.000,C 90.000,E1 164.102} C_DIS
LIN {X 0.066,Y -150.098,Z 690.891,A 0.000,B 0.000,C 90.000,E1 160.423} C_DIS
LIN {X 0.078,Y -153.453,Z 690.871,A 0.000,B 0.000,C 90.000,E1 156.794} C_DIS
LIN {X -0.070,Y -157.816,Z 690.846,A 0.000,B 0.000,C 90.000,E1 152.359} C_DIS
LIN {X -0.038,Y -162.099,Z 690.827,A 0.000,B 0.000,C 90.000,E1 148.791} C_DIS
LIN {X -0.014,Y -166.299,Z 690.807,A 0.000,B 0.000,C 90.000,E1 145.261} C_DIS
LIN {X -0.016,Y -171.316,Z 690.788,A 0.000,B 0.000,C 90.000,E1 141.778} C_DIS
LIN {X 0.018,Y -176.215,Z 690.768,A 0.000,B 0.000,C 90.000,E1 138.324} C_DIS
LIN {X 0.011,Y -180.492,Z 690.754,A 0.000,B 0.000,C 90.000,E1 135.769} C_DIS
LIN {X -0.007,Y -185.896,Z 690.736,A 0.000,B 0.000,C 90.000,E1 132.405} C_DIS
LIN {X -0.006,Y -191.248,Z 690.719,A 0.000,B 0.000,C 90.000,E1 129.483} C_DIS
LIN {X -0.043,Y -288.665,Z 690.719,A 0.000,B 0.000,C 90.000,E1 129.483} C_DIS
LIN {X 0.008,Y -291.160,Z 690.719,A 0.000,B 0.000,C 90.000,E1 129.439} C_DIS
LIN {X -0.102,Y -295.138,Z 690.718,A 0.000,B 0.000,C 90.000,E1 129.277} C_DIS
LIN {X 0.017,Y -297.419,Z 690.717,A 0.000,B 0.000,C 90.000,E1 129.072} C_DIS
LIN {X 0.069,Y -301.284,Z 690.714,A 0.000,B 0.000,C 90.000,E1 128.588} C_DIS
LIN {X 0.075,Y -303.146,Z 690.713,A 0.000,B 0.000,C 90.000,E1 128.257} C_DIS
LIN {X 0.031,Y -304.600,Z 690.711,A 0.000,B 0.000,C 90.000,E1 127.935} C_DIS
LIN {X 0.004,Y -306.663,Z 690.707,A 0.000,B 0.000,C 90.000,E1 127.282} C_DIS
LIN {X -0.070,Y -316.362,Z 690.689,A 0.000,B 0.000,C 90.000,E1 124.040} C_DIS
LIN {X 0.100,Y -326.384,Z 690.673,A 0.000,B 0.000,C 90.000,E1 121.131} C_DIS
LIN {X 0.071,Y -337.735,Z 690.657,A 0.000,B 0.000,C 90.000,E1 118.309} C_DIS
LIN {X 0.059,Y -350.509,Z 690.642,A 0.000,B 0.000,C 90.000,E1 115.540} C_DIS
LIN {X 0.031,Y -363.155,Z 690.629,A 0.000,B 0.000,C 90.000,E1 113.131} C_DIS
LIN {X -0.118,Y -377.110,Z 690.615,A 0.000,B 0.000,C 90.000,E1 110.791} C_DIS
LIN {X -0.056,Y -392.473,Z 690.603,A 0.000,B 0.000,C 90.000,E1 108.471} C_DIS
LIN {X 0.028,Y -409.357,Z 690.590,A 0.000,B 0.000,C 90.000,E1 106.205} C_DIS
LIN {X 0.037,Y -427.884,Z 690.578,A 0.000,B 0.000,C 90.000,E1 104.008} C_DIS
LIN {X -0.250,Y -447.783,Z 690.566,A 0.000,B 0.000,C 90.000,E1 101.951} C_DIS
LIN {X -0.184,Y -468.282,Z 690.556,A 0.000,B 0.000,C 90.000,E1 100.018} C_DIS
LIN {X -0.141,Y -470.516,Z 690.554,A 0.000,B 0.000,C 90.000,E1 99.782} C_DIS
LIN {X 0.110,Y -472.340,Z 690.553,A 0.000,B 0.000,C 90.000,E1 99.500} C_DIS
LIN {X -0.026,Y -473.712,Z 690.551,A 0.000,B 0.000,C 90.000,E1 99.265} C_DIS
LIN {X 0.088,Y -475.458,Z 690.549,A 0.000,B 0.000,C 90.000,E1 98.746} C_DIS
LIN {X -0.190,Y -476.124,Z 690.546,A 0.000,B 0.000,C 90.000,E1 98.276} C_DIS
LIN {X -0.058,Y -475.821,Z 690.543,A 0.000,B 0.000,C 90.000,E1 97.757} C_DIS
LIN {X 0.080,Y -474.508,Z 690.540,A 0.000,B 0.000,C 90.000,E1 97.239} C_DIS
LIN {X -0.058,Y -473.409,Z 690.539,A 0.000,B 0.000,C 90.000,E1 97.004} C_DIS
LIN {X 0.215,Y -471.938,Z 690.537,A 0.000,B 0.000,C 90.000,E1 96.720} C_DIS
LIN {X -0.079,Y -453.693,Z 690.522,A 0.000,B 0.000,C 90.000,E1 93.955} C_DIS
LIN {X -0.104,Y -437.484,Z 690.506,A 0.000,B 0.000,C 90.000,E1 91.088} C_DIS
LIN {X -0.025,Y -428.587,Z 690.497,A 0.000,B 0.000,C 90.000,E1 89.484} C_DIS
LIN {X -0.093,Y -419.306,Z 690.488,A 0.000,B 0.000,C 90.000,E1 87.879} C_DIS
LIN {X 0.163,Y -408.357,Z 690.478,A 0.000,B 0.000,C 90.000,E1 85.931} C_DIS
LIN {X -0.090,Y -395.849,Z 690.465,A 0.000,B 0.000,C 90.000,E1 83.742} C_DIS
LIN {X -0.113,Y -380.647,Z 690.449,A 0.000,B 0.000,C 90.000,E1 80.905} C_DIS
LIN {X -0.070,Y -368.953,Z 690.436,A 0.000,B 0.000,C 90.000,E1 78.578} C_DIS
LIN {X 0.133,Y -353.487,Z 690.418,A 0.000,B 0.000,C 90.000,E1 75.283} C_DIS
LIN {X -0.149,Y -341.452,Z 690.403,A 0.000,B 0.000,C 90.000,E1 72.598} C_DIS
LIN {X 0.060,Y -328.649,Z 690.386,A 0.000,B 0.000,C 90.000,E1 69.464} C_DIS
LIN {X 0.086,Y -315.791,Z 690.367,A 0.000,B 0.000,C 90.000,E1 65.973} C_DIS
LIN {X 0.017,Y -303.646,Z 690.345,A 0.000,B 0.000,C 90.000,E1 62.103} C_DIS
LIN {X 0.089,Y -294.444,Z 690.327,A 0.000,B 0.000,C 90.000,E1 58.791} C_DIS
LIN {X -0.064,Y -285.865,Z 690.308,A 0.000,B 0.000,C 90.000,E1 55.468} C_DIS
LIN {X 0.082,Y -279.201,Z 690.293,A 0.000,B 0.000,C 90.000,E1 52.718} C_DIS
LIN {X -0.032,Y -274.060,Z 690.281,A 0.000,B 0.000,C 90.000,E1 50.678} C_DIS
LIN {X -0.095,Y -268.695,Z 690.270,A 0.000,B 0.000,C 90.000,E1 48.609} C_DIS
LIN {X 0.121,Y -262.955,Z 690.258,A 0.000,B 0.000,C 90.000,E1 46.458} C_DIS
LIN {X 0.025,Y -256.960,Z 690.246,A 0.000,B 0.000,C 90.000,E1 44.352} C_DIS
LIN {X 0.002,Y -250.877,Z 690.234,A 0.000,B 0.000,C 90.000,E1 42.204} C_DIS
LIN {X 0.065,Y -244.636,Z 690.222,A 0.000,B 0.000,C 90.000,E1 40.011} C_DIS
LIN {X 0.013,Y -236.382,Z 690.206,A 0.000,B 0.000,C 90.000,E1 37.076} C_DIS
LIN {X 0.132,Y -226.765,Z 690.185,A 0.000,B 0.000,C 90.000,E1 33.293} C_DIS
LIN {X 0.053,Y -219.915,Z 690.168,A 0.000,B 0.000,C 90.000,E1 30.256} C_DIS
LIN {X -0.032,Y -213.847,Z 690.151,A 0.000,B 0.000,C 90.000,E1 27.180} C_DIS
LIN {X 0.021,Y -208.600,Z 690.133,A 0.000,B 0.000,C 90.000,E1 24.027} C_DIS
LIN {X -0.022,Y -203.201,Z 690.111,A 0.000,B 0.000,C 90.000,E1 20.066} C_DIS
LIN {X 0.066,Y -198.991,Z 690.089,A 0.000,B 0.000,C 90.000,E1 16.024} C_DIS
LIN {X -0.032,Y -195.339,Z 690.062,A 0.000,B 0.000,C 90.000,E1 11.186} C_DIS
LIN {X -0.032,Y -192.770,Z 690.026,A 0.000,B 0.000,C 90.000,E1 4.645} C_DIS
LIN {X -0.033,Y -194.198,Z 689.966,A 0.000,B 0.000,C 90.000,E1 353.799} C_DIS
LIN {X 0.090,Y -197.781,Z 689.934,A 0.000,B 0.000,C 90.000,E1 348.049} C_DIS
LIN {X -0.023,Y -201.528,Z 689.911,A 0.000,B 0.000,C 90.000,E1 344.031} C_DIS
LIN {X 0.005,Y -206.229,Z 689.889,A 0.000,B 0.000,C 90.000,E1 340.007} C_DIS
LIN {X -0.052,Y -211.780,Z 689.867,A 0.000,B 0.000,C 90.000,E1 336.049} C_DIS
LIN {X 0.027,Y -217.994,Z 689.845,A 0.000,B 0.000,C 90.000,E1 332.103} C_DIS
LIN {X -0.049,Y -225.000,Z 689.824,A 0.000,B 0.000,C 90.000,E1 328.250} C_DIS
LIN {X 0.082,Y -232.558,Z 689.802,A 0.000,B 0.000,C 90.000,E1 324.402} C_DIS
LIN {X 0.107,Y -240.786,Z 689.781,A 0.000,B 0.000,C 90.000,E1 320.642} C_DIS
LIN {X -0.044,Y -249.910,Z 689.761,A 0.000,B 0.000,C 90.000,E1 316.986} C_DIS
LIN {X 0.055,Y -259.069,Z 689.743,A 0.000,B 0.000,C 90.000,E1 313.704} C_DIS
LIN {X -0.030,Y -270.320,Z 689.723,A 0.000,B 0.000,C 90.000,E1 310.172} C_DIS
LIN {X 0.035,Y -281.648,Z 689.706,A 0.000,B 0.000,C 90.000,E1 307.030} C_DIS
LIN {X 0.076,Y -295.544,Z 689.687,A 0.000,B 0.000,C 90.000,E1 303.627} C_DIS
LIN {X -0.010,Y -310.876,Z 689.669,A 0.000,B 0.000,C 90.000,E1 300.335} C_DIS
LIN {X -0.073,Y -327.801,Z 689.651,A 0.000,B 0.000,C 90.000,E1 297.129} C_DIS
LIN {X -0.194,Y -344.056,Z 689.635,A 0.000,B 0.000,C 90.000,E1 294.335} C_DIS
LIN {X -0.089,Y -363.269,Z 689.618,A 0.000,B 0.000,C 90.000,E1 291.280} C_DIS
LIN {X -0.088,Y -375.521,Z 689.608,A 0.000,B 0.000,C 90.000,E1 289.504} C_DIS
LIN {X 0.038,Y -391.233,Z 689.597,A 0.000,B 0.000,C 90.000,E1 287.457} C_DIS
LIN {X -0.172,Y -405.267,Z 689.588,A 0.000,B 0.000,C 90.000,E1 285.788} C_DIS
LIN {X -0.134,Y -419.041,Z 689.578,A 0.000,B 0.000,C 90.000,E1 284.120} C_DIS
LIN {X -0.218,Y -430.154,Z 689.571,A 0.000,B 0.000,C 90.000,E1 282.771} C_DIS
LIN {X 0.092,Y -438.675,Z 689.565,A 0.000,B 0.000,C 90.000,E1 281.658} C_DIS
LIN {X 0.077,Y -446.725,Z 689.559,A 0.000,B 0.000,C 90.000,E1 280.602} C_DIS
LIN {X -0.018,Y -464.768,Z 689.546,A 0.000,B 0.000,C 90.000,E1 278.276} C_DIS
LIN {X -0.184,Y -470.640,Z 689.542,A 0.000,B 0.000,C 90.000,E1 277.530} C_DIS
LIN {X 0.231,Y -475.943,Z 689.537,A 0.000,B 0.000,C 90.000,E1 276.720} C_DIS
LIN {X -0.114,Y -478.975,Z 689.535,A 0.000,B 0.000,C 90.000,E1 276.258} C_DIS
LIN {X -0.147,Y -482.693,Z 689.531,A 0.000,B 0.000,C 90.000,E1 275.511} C_DIS
LIN {X -0.106,Y -485.373,Z 689.526,A 0.000,B 0.000,C 90.000,E1 274.759} C_DIS
LIN {X 0.038,Y -486.657,Z 689.524,A 0.000,B 0.000,C 90.000,E1 274.245} C_DIS
LIN {X 0.231,Y -487.512,Z 689.521,A 0.000,B 0.000,C 90.000,E1 273.726} C_DIS
LIN {X -0.088,Y -488.056,Z 689.518,A 0.000,B 0.000,C 90.000,E1 273.269} C_DIS
LIN {X 0.114,Y -488.229,Z 689.515,A 0.000,B 0.000,C 90.000,E1 272.751} C_DIS
LIN {X -0.194,Y -488.078,Z 689.513,A 0.000,B 0.000,C 90.000,E1 272.293} C_DIS
LIN {X 0.006,Y -487.601,Z 689.510,A 0.000,B 0.000,C 90.000,E1 271.776} C_DIS
LIN {X 0.186,Y -486.793,Z 689.507,A 0.000,B 0.000,C 90.000,E1 271.260} C_DIS
LIN {X -0.120,Y -485.579,Z 689.504,A 0.000,B 0.000,C 90.000,E1 270.802} C_DIS
LIN {X 0.056,Y -483.868,Z 689.502,A 0.000,B 0.000,C 90.000,E1 270.286} C_DIS
LIN {X 0.223,Y -481.592,Z 689.499,A 0.000,B 0.000,C 90.000,E1 269.771} C_DIS
LIN {X -0.107,Y -478.660,Z 689.496,A 0.000,B 0.000,C 90.000,E1 269.312} C_DIS
LIN {X 0.029,Y -474.959,Z 689.493,A 0.000,B 0.000,C 90.000,E1 268.797} C_DIS
LIN {X 0.142,Y -470.245,Z 689.491,A 0.000,B 0.000,C 90.000,E1 268.282} C_DIS
LIN {X -0.017,Y -467.475,Z 689.489,A 0.000,B 0.000,C 90.000,E1 268.051} C_DIS
LIN {X -0.070,Y -461.339,Z 689.487,A 0.000,B 0.000,C 90.000,E1 267.593} C_DIS
LIN {X 0.020,Y -454.597,Z 689.484,A 0.000,B 0.000,C 90.000,E1 267.192} C_DIS
LIN {X -0.226,Y -447.618,Z 689.483,A 0.000,B 0.000,C 90.000,E1 266.906} C_DIS
LIN {X 0.023,Y -440.385,Z 689.481,A 0.000,B 0.000,C 90.000,E1 266.617} C_DIS
LIN {X 0.021,Y -436.308,Z 689.481,A 0.000,B 0.000,C 90.000,E1 266.502} C_DIS
LIN {X -0.212,Y -432.228,Z 689.480,A 0.000,B 0.000,C 90.000,E1 266.445} C_DIS
LIN {X 0.075,Y -421.738,Z 689.479,A 0.000,B 0.000,C 90.000,E1 266.274} C_DIS
LIN {X -0.169,Y -415.696,Z 689.479,A 0.000,B 0.000,C 90.000,E1 266.274} C_DIS
LIN {X 0.086,Y -180.932,Z 689.479,A 0.000,B 0.000,C 90.000,E1 266.216} C_DIS
LIN {X -0.037,Y -180.772,Z 689.471,A 0.000,B 0.000,C 90.000,E1 264.723} C_DIS
LIN {X 0.000,Y -178.988,Z 689.444,A 0.000,B 0.000,C 90.000,E1 259.982} C_DIS
LIN {X 0.011,Y -177.970,Z 689.435,A 0.000,B 0.000,C 90.000,E1 258.285} C_DIS
LIN {X 0.030,Y -175.612,Z 689.411,A 0.000,B 0.000,C 90.000,E1 254.031} C_DIS
LIN {X 0.042,Y -172.334,Z 689.388,A 0.000,B 0.000,C 90.000,E1 249.752} C_DIS
LIN {X 0.021,Y -171.812,Z 689.383,A 0.000,B 0.000,C 90.000,E1 248.901} C_DIS
LIN {X 0.028,Y -170.275,Z 689.373,A 0.000,B 0.000,C 90.000,E1 247.177} C_DIS
LIN {X -0.035,Y -166.816,Z 689.349,A 0.000,B 0.000,C 90.000,E1 242.871} C_DIS
LIN {X 0.021,Y -162.798,Z 689.325,A 0.000,B 0.000,C 90.000,E1 238.486} C_DIS
LIN {X -0.054,Y -161.485,Z 689.315,A 0.000,B 0.000,C 90.000,E1 236.755} C_DIS
LIN {X -0.003,Y -157.481,Z 689.291,A 0.000,B 0.000,C 90.000,E1 232.316} C_DIS
LIN {X 0.054,Y -155.498,Z 689.276,A 0.000,B 0.000,C 90.000,E1 229.622} C_DIS
LIN {X -0.014,Y -151.802,Z 689.251,A 0.000,B 0.000,C 90.000,E1 225.162} C_DIS
LIN {X -0.001,Y -150.012,Z 689.236,A 0.000,B 0.000,C 90.000,E1 222.447} C_DIS
LIN {X 0.030,Y -146.837,Z 689.211,A 0.000,B 0.000,C 90.000,E1 217.890} C_DIS
LIN {X 0.016,Y -145.419,Z 689.195,A 0.000,B 0.000,C 90.000,E1 215.152} C_DIS
LIN {X 0.052,Y -142.846,Z 689.170,A 0.000,B 0.000,C 90.000,E1 210.541} C_DIS
LIN {X -0.018,Y -141.461,Z 689.149,A 0.000,B 0.000,C 90.000,E1 206.873} C_DIS
LIN {X 0.021,Y -139.375,Z 689.113,A 0.000,B 0.000,C 90.000,E1 200.355} C_DIS
LIN {X -0.037,Y -138.826,Z 689.098,A 0.000,B 0.000,C 90.000,E1 197.583} C_DIS
LIN {X 0.051,Y -138.353,Z 689.056,A 0.000,B 0.000,C 90.000,E1 190.074} C_DIS
LIN {X 0.025,Y -139.530,Z 689.004,A 0.000,B 0.000,C 90.000,E1 180.745} C_DIS
LIN {X -0.022,Y -141.208,Z 688.973,A 0.000,B 0.000,C 90.000,E1 175.179} C_DIS
LIN {X -0.064,Y -142.584,Z 688.958,A 0.000,B 0.000,C 90.000,E1 172.413} C_DIS
LIN {X 0.032,Y -144.879,Z 688.932,A 0.000,B 0.000,C 90.000,E1 167.757} C_DIS
LIN {X -0.014,Y -147.507,Z 688.912,A 0.000,B 0.000,C 90.000,E1 164.102} C_DIS
LIN {X 0.061,Y -150.098,Z 688.891,A 0.000,B 0.000,C 90.000,E1 160.423} C_DIS
LIN {X 0.073,Y -153.455,Z 688.871,A 0.000,B 0.000,C 90.000,E1 156.794} C_DIS
LIN {X -0.075,Y -157.817,Z 688.846,A 0.000,B 0.000,C 90.000,E1 152.359} C_DIS
LIN {X -0.043,Y -162.101,Z 688.827,A 0.000,B 0.000,C 90.000,E1 148.791} C_DIS
LIN {X -0.018,Y -166.301,Z 688.807,A 0.000,B 0.000,C 90.000,E1 145.261} C_DIS
LIN {X -0.022,Y -171.318,Z 688.788,A 0.000,B 0.000,C 90.000,E1 141.778} C_DIS
LIN {X 0.013,Y -176.217,Z 688.768,A 0.000,B 0.000,C 90.000,E1 138.324} C_DIS
LIN {X 0.006,Y -180.495,Z 688.754,A 0.000,B 0.000,C 90.000,E1 135.769} C_DIS
LIN {X -0.012,Y -185.898,Z 688.736,A 0.000,B 0.000,C 90.000,E1 132.405} C_DIS
LIN {X 0.013,Y -191.239,Z 688.719,A 0.000,B 0.000,C 90.000,E1 129.483} C_DIS
LIN {X -0.015,Y -289.623,Z 688.719,A 0.000,B 0.000,C 90.000,E1 129.483} C_DIS
LIN {X 0.002,Y -291.579,Z 688.719,A 0.000,B 0.000,C 90.000,E1 129.439} C_DIS
LIN {X -0.109,Y -295.282,Z 688.718,A 0.000,B 0.000,C 90.000,E1 129.277} C_DIS
LIN {X 0.009,Y -297.509,Z 688.717,A 0.000,B 0.000,C 90.000,E1 129.072} C_DIS
LIN {X 0.008,Y -301.381,Z 688.714,A 0.000,B 0.000,C 90.000,E1 128.588} C_DIS
LIN {X 0.003,Y -303.220,Z 688.713,A 0.000,B 0.000,C 90.000,E1 128.257} C_DIS
LIN {X -0.054,Y -304.656,Z 688.711,A 0.000,B 0.000,C 90.000,E1 127.935} C_DIS
LIN {X -0.080,Y -306.686,Z 688.707,A 0.000,B 0.000,C 90.000,E1 127.282} C_DIS
LIN {X 0.105,Y -316.392,Z 688.689,A 0.000,B 0.000,C 90.000,E1 123.992} C_DIS
LIN {X 0.011,Y -326.421,Z 688.673,A 0.000,B 0.000,C 90.000,E1 121.131} C_DIS
LIN {X -0.019,Y -337.779,Z 688.657,A 0.000,B 0.000,C 90.000,E1 118.309} C_DIS
LIN {X -0.035,Y -350.561,Z 688.642,A 0.000,B 0.000,C 90.000,E1 115.540} C_DIS
LIN {X -0.064,Y -363.216,Z 688.628,A 0.000,B 0.000,C 90.000,E1 113.131} C_DIS
LIN {X 0.137,Y -377.178,Z 688.615,A 0.000,B 0.000,C 90.000,E1 110.737} C_DIS
LIN {X 0.216,Y -392.551,Z 688.602,A 0.000,B 0.000,C 90.000,E1 108.417} C_DIS
LIN {X -0.075,Y -409.444,Z 688.590,A 0.000,B 0.000,C 90.000,E1 106.205} C_DIS
LIN {X -0.067,Y -427.982,Z 688.578,A 0.000,B 0.000,C 90.000,E1 104.008} C_DIS
LIN {X 0.088,Y -447.886,Z 688.566,A 0.000,B 0.000,C 90.000,E1 101.895} C_DIS
LIN {X 0.179,Y -468.387,Z 688.555,A 0.000,B 0.000,C 90.000,E1 99.962} C_DIS
LIN {X 0.225,Y -470.608,Z 688.554,A 0.000,B 0.000,C 90.000,E1 99.726} C_DIS
LIN {X 0.005,Y -472.429,Z 688.553,A 0.000,B 0.000,C 90.000,E1 99.500} C_DIS
LIN {X -0.137,Y -473.797,Z 688.551,A 0.000,B 0.000,C 90.000,E1 99.265} C_DIS
LIN {X -0.024,Y -475.529,Z 688.549,A 0.000,B 0.000,C 90.000,E1 98.746} C_DIS
LIN {X 0.169,Y -476.183,Z 688.546,A 0.000,B 0.000,C 90.000,E1 98.219} C_DIS
LIN {X -0.169,Y -475.869,Z 688.543,A 0.000,B 0.000,C 90.000,E1 97.757} C_DIS
LIN {X -0.031,Y -474.543,Z 688.540,A 0.000,B 0.000,C 90.000,E1 97.239} C_DIS
LIN {X -0.169,Y -473.437,Z 688.539,A 0.000,B 0.000,C 90.000,E1 97.004} C_DIS
LIN {X 0.107,Y -471.957,Z 688.537,A 0.000,B 0.000,C 90.000,E1 96.720} C_DIS
LIN {X -0.184,Y -453.698,Z 688.522,A 0.000,B 0.000,C 90.000,E1 93.955} C_DIS
LIN {X -0.204,Y -437.494,Z 688.506,A 0.000,B 0.000,C 90.000,E1 91.088} C_DIS
LIN {X 0.159,Y -430.122,Z 688.499,A 0.000,B 0.000,C 90.000,E1 89.714} C_DIS
LIN {X 0.113,Y -420.882,Z 688.490,A 0.000,B 0.000,C 90.000,E1 88.108} C_DIS
LIN {X -0.003,Y -409.966,Z 688.479,A 0.000,B 0.000,C 90.000,E1 86.216} C_DIS
LIN {X 0.107,Y -398.969,Z 688.468,A 0.000,B 0.000,C 90.000,E1 84.261} C_DIS
LIN {X 0.073,Y -385.193,Z 688.454,A 0.000,B 0.000,C 90.000,E1 81.724} C_DIS
LIN {X -0.157,Y -373.377,Z 688.441,A 0.000,B 0.000,C 90.000,E1 79.454} C_DIS
LIN {X 0.131,Y -361.866,Z 688.428,A 0.000,B 0.000,C 90.000,E1 77.061} C_DIS
LIN {X -0.032,Y -349.537,Z 688.413,A 0.000,B 0.000,C 90.000,E1 74.393} C_DIS
LIN {X 0.006,Y -336.376,Z 688.396,A 0.000,B 0.000,C 90.000,E1 71.329} C_DIS
LIN {X -0.061,Y -322.782,Z 688.377,A 0.000,B 0.000,C 90.000,E1 67.901} C_DIS
LIN {X -0.122,Y -311.752,Z 688.359,A 0.000,B 0.000,C 90.000,E1 64.717} C_DIS
LIN {X 0.039,Y -301.948,Z 688.341,A 0.000,B 0.000,C 90.000,E1 61.435} C_DIS
LIN {X 0.063,Y -292.913,Z 688.323,A 0.000,B 0.000,C 90.000,E1 58.122} C_DIS
LIN {X 0.018,Y -284.449,Z 688.304,A 0.000,B 0.000,C 90.000,E1 54.769} C_DIS
LIN {X 0.074,Y -277.810,Z 688.289,A 0.000,B 0.000,C 90.000,E1 52.029} C_DIS
LIN {X -0.059,Y -272.587,Z 688.278,A 0.000,B 0.000,C 90.000,E1 49.989} C_DIS
LIN {X 0.053,Y -267.080,Z 688.266,A 0.000,B 0.000,C 90.000,E1 47.877} C_DIS
LIN {X -0.151,Y -261.227,Z 688.254,A 0.000,B 0.000,C 90.000,E1 45.810} C_DIS
LIN {X 0.089,Y -255.192,Z 688.242,A 0.000,B 0.000,C 90.000,E1 43.623} C_DIS
LIN {X 0.047,Y -249.032,Z 688.230,A 0.000,B 0.000,C 90.000,E1 41.472} C_DIS
LIN {X 0.080,Y -242.727,Z 688.218,A 0.000,B 0.000,C 90.000,E1 39.277} C_DIS
LIN {X -0.029,Y -232.609,Z 688.198,A 0.000,B 0.000,C 90.000,E1 35.598} C_DIS
LIN {X 0.100,Y -225.135,Z 688.181,A 0.000,B 0.000,C 90.000,E1 32.546} C_DIS
LIN {X -0.128,Y -218.522,Z 688.164,A 0.000,B 0.000,C 90.000,E1 29.539} C_DIS
LIN {X -0.054,Y -212.638,Z 688.147,A 0.000,B 0.000,C 90.000,E1 26.411} C_DIS
LIN {X -0.032,Y -207.604,Z 688.129,A 0.000,B 0.000,C 90.000,E1 23.259} C_DIS
LIN {X 0.004,Y -202.443,Z 688.107,A 0.000,B 0.000,C 90.000,E1 19.268} C_DIS
LIN {X 0.004,Y -198.441,Z 688.085,A 0.000,B 0.000,C 90.000,E1 15.245} C_DIS
LIN {X 0.028,Y -195.031,Z 688.058,A 0.000,B 0.000,C 90.000,E1 10.366} C_DIS
LIN {X -0.091,Y -192.696,Z 688.017,A 0.000,B 0.000,C 90.000,E1 3.037} C_DIS
